REGION Network 3: Перше слово повідомлень
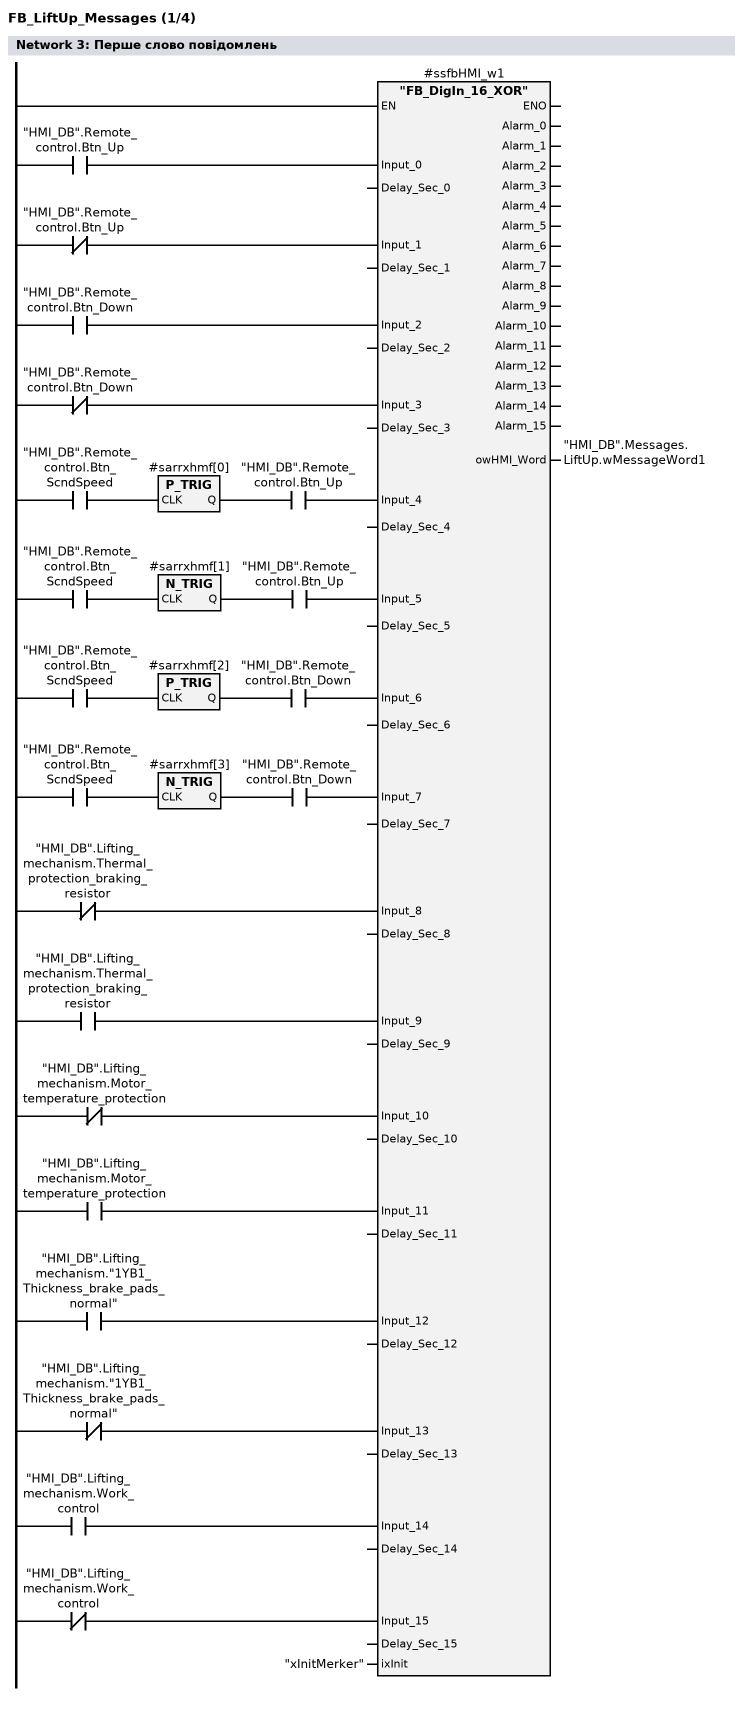
   RUNG wire#powerrail
      #ssfbHMI_w1(Input_0 := wire#w1, Input_1 := wire#w2, Input_2 := wire#w3, Input_3 := wire#w4, Input_4 := wire#w5, Input_5 := wire#w6, Input_6 := wire#w7, Input_7 := wire#w8, Input_8 := wire#w9, Input_9 := wire#w10, Input_10 := wire#w11, Input_11 := wire#w12, Input_12 := wire#w13, Input_13 := wire#w14, Input_14 := wire#w15, Input_15 := wire#w16, Delay_Sec_0 :=, Delay_Sec_1 :=, Delay_Sec_2 :=, Delay_Sec_3 :=, Delay_Sec_4 :=, Delay_Sec_5 :=, Delay_Sec_6 :=, Delay_Sec_7 :=, Delay_Sec_8 :=, Delay_Sec_9 :=, Delay_Sec_10 :=, Delay_Sec_11 :=, Delay_Sec_12 :=, Delay_Sec_13 :=, Delay_Sec_14 :=, Delay_Sec_15 :=, ixInit := "xInitMerker", Alarm_0 =>, Alarm_1 =>, Alarm_2 =>, Alarm_3 =>, Alarm_4 =>, Alarm_5 =>, Alarm_6 =>, Alarm_7 =>, Alarm_8 =>, Alarm_9 =>, Alarm_10 =>, Alarm_11 =>, Alarm_12 =>, Alarm_13 =>, Alarm_14 =>, Alarm_15 =>, owHMI_Word => "HMI_DB".Messages.LiftUp.wMessageWord1)
   END_RUNG
   RUNG wire#powerrail
      Contact( "HMI_DB".Remote_control.Btn_Up )
   END_RUNG wire#w1
   RUNG wire#powerrail
      I_Contact( "HMI_DB".Remote_control.Btn_Up )
   END_RUNG wire#w2
   RUNG wire#powerrail
      Contact( "HMI_DB".Remote_control.Btn_Down )
   END_RUNG wire#w3
   RUNG wire#powerrail
      I_Contact( "HMI_DB".Remote_control.Btn_Down )
   END_RUNG wire#w4
   RUNG wire#powerrail
      Contact( "HMI_DB".Remote_control.Btn_ScndSpeed )
      P_Trig( #sarrxhmf[0] )
      Contact( "HMI_DB".Remote_control.Btn_Up )
   END_RUNG wire#w5
   RUNG wire#powerrail
      Contact( "HMI_DB".Remote_control.Btn_ScndSpeed )
      N_Trig( #sarrxhmf[1] )
      Contact( "HMI_DB".Remote_control.Btn_Up )
   END_RUNG wire#w6
   RUNG wire#powerrail
      Contact( "HMI_DB".Remote_control.Btn_ScndSpeed )
      P_Trig( #sarrxhmf[2] )
      Contact( "HMI_DB".Remote_control.Btn_Down )
   END_RUNG wire#w7
   RUNG wire#powerrail
      Contact( "HMI_DB".Remote_control.Btn_ScndSpeed )
      N_Trig( #sarrxhmf[3] )
      Contact( "HMI_DB".Remote_control.Btn_Down )
   END_RUNG wire#w8
   RUNG wire#powerrail
      I_Contact( "HMI_DB".Lifting_mechanism.Thermal_protection_braking_resistor )
   END_RUNG wire#w9
   RUNG wire#powerrail
      Contact( "HMI_DB".Lifting_mechanism.Thermal_protection_braking_resistor )
   END_RUNG wire#w10
   RUNG wire#powerrail
      I_Contact( "HMI_DB".Lifting_mechanism.Motor_temperature_protection )
   END_RUNG wire#w11
   RUNG wire#powerrail
      Contact( "HMI_DB".Lifting_mechanism.Motor_temperature_protection )
   END_RUNG wire#w12
   RUNG wire#powerrail
      Contact( "HMI_DB".Lifting_mechanism."1YB1_Thickness_brake_pads_normal" )
   END_RUNG wire#w13
   RUNG wire#powerrail
      I_Contact( "HMI_DB".Lifting_mechanism."1YB1_Thickness_brake_pads_normal" )
   END_RUNG wire#w14
   RUNG wire#powerrail
      Contact( "HMI_DB".Lifting_mechanism.Work_control )
   END_RUNG wire#w15
   RUNG wire#powerrail
      I_Contact( "HMI_DB".Lifting_mechanism.Work_control )
   END_RUNG wire#w16
   // the same network as SCL:
   #_w1 := "HMI_DB".Remote_control.Btn_ScndSpeed AND NOT #sarrxhmf[0];   // rising edge
   #sarrxhmf[0] := "HMI_DB".Remote_control.Btn_ScndSpeed;
   #_w2 := NOT "HMI_DB".Remote_control.Btn_ScndSpeed AND #sarrxhmf[1];   // falling edge
   #sarrxhmf[1] := "HMI_DB".Remote_control.Btn_ScndSpeed;
   #_w3 := "HMI_DB".Remote_control.Btn_ScndSpeed AND NOT #sarrxhmf[2];   // rising edge
   #sarrxhmf[2] := "HMI_DB".Remote_control.Btn_ScndSpeed;
   #_w4 := NOT "HMI_DB".Remote_control.Btn_ScndSpeed AND #sarrxhmf[3];   // falling edge
   #sarrxhmf[3] := "HMI_DB".Remote_control.Btn_ScndSpeed;
   #ssfbHMI_w1(Input_0 := "HMI_DB".Remote_control.Btn_Up,   // "FB_DigIn_16_XOR"
               Input_1 := NOT "HMI_DB".Remote_control.Btn_Up,
               Input_2 := "HMI_DB".Remote_control.Btn_Down,
               Input_3 := NOT "HMI_DB".Remote_control.Btn_Down,
               Input_4 := #_w1 AND "HMI_DB".Remote_control.Btn_Up,
               Input_5 := #_w2 AND "HMI_DB".Remote_control.Btn_Up,
               Input_6 := #_w3 AND "HMI_DB".Remote_control.Btn_Down,
               Input_7 := #_w4 AND "HMI_DB".Remote_control.Btn_Down,
               Input_8 := NOT "HMI_DB".Lifting_mechanism.Thermal_protection_braking_resistor,
               Input_9 := "HMI_DB".Lifting_mechanism.Thermal_protection_braking_resistor,
               Input_10 := NOT "HMI_DB".Lifting_mechanism.Motor_temperature_protection,
               Input_11 := "HMI_DB".Lifting_mechanism.Motor_temperature_protection,
               Input_12 := "HMI_DB".Lifting_mechanism."1YB1_Thickness_brake_pads_normal",
               Input_13 := NOT "HMI_DB".Lifting_mechanism."1YB1_Thickness_brake_pads_normal",
               Input_14 := "HMI_DB".Lifting_mechanism.Work_control,
               Input_15 := NOT "HMI_DB".Lifting_mechanism.Work_control,
               ixInit := "xInitMerker",
               owHMI_Word => "HMI_DB".Messages.LiftUp.wMessageWord1);
END_REGION

REGION Network 4: Друге слово повідомлень
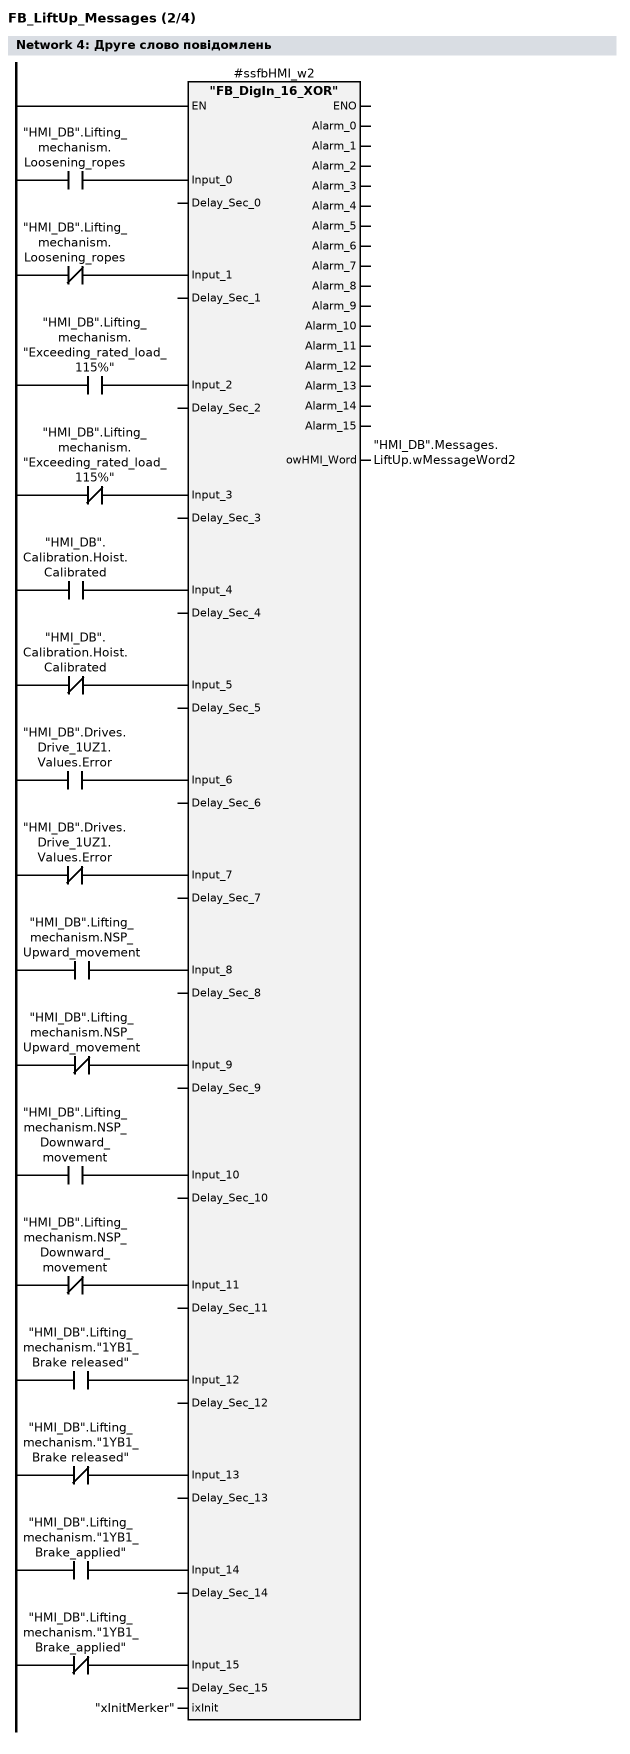
   RUNG wire#powerrail
      #ssfbHMI_w2(Input_0 := wire#w1, Input_1 := wire#w2, Input_2 := wire#w3, Input_3 := wire#w4, Input_4 := wire#w5, Input_5 := wire#w6, Input_6 := wire#w7, Input_7 := wire#w8, Input_8 := wire#w9, Input_9 := wire#w10, Input_10 := wire#w11, Input_11 := wire#w12, Input_12 := wire#w13, Input_13 := wire#w14, Input_14 := wire#w15, Input_15 := wire#w16, Delay_Sec_0 :=, Delay_Sec_1 :=, Delay_Sec_2 :=, Delay_Sec_3 :=, Delay_Sec_4 :=, Delay_Sec_5 :=, Delay_Sec_6 :=, Delay_Sec_7 :=, Delay_Sec_8 :=, Delay_Sec_9 :=, Delay_Sec_10 :=, Delay_Sec_11 :=, Delay_Sec_12 :=, Delay_Sec_13 :=, Delay_Sec_14 :=, Delay_Sec_15 :=, ixInit := "xInitMerker", Alarm_0 =>, Alarm_1 =>, Alarm_2 =>, Alarm_3 =>, Alarm_4 =>, Alarm_5 =>, Alarm_6 =>, Alarm_7 =>, Alarm_8 =>, Alarm_9 =>, Alarm_10 =>, Alarm_11 =>, Alarm_12 =>, Alarm_13 =>, Alarm_14 =>, Alarm_15 =>, owHMI_Word => "HMI_DB".Messages.LiftUp.wMessageWord2)
   END_RUNG
   RUNG wire#powerrail
      Contact( "HMI_DB".Lifting_mechanism.Loosening_ropes )
   END_RUNG wire#w1
   RUNG wire#powerrail
      I_Contact( "HMI_DB".Lifting_mechanism.Loosening_ropes )
   END_RUNG wire#w2
   RUNG wire#powerrail
      Contact( "HMI_DB".Lifting_mechanism."Exceeding_rated_load_115%" )
   END_RUNG wire#w3
   RUNG wire#powerrail
      I_Contact( "HMI_DB".Lifting_mechanism."Exceeding_rated_load_115%" )
   END_RUNG wire#w4
   RUNG wire#powerrail
      Contact( "HMI_DB".Calibration.Hoist.Calibrated )
   END_RUNG wire#w5
   RUNG wire#powerrail
      I_Contact( "HMI_DB".Calibration.Hoist.Calibrated )
   END_RUNG wire#w6
   RUNG wire#powerrail
      Contact( "HMI_DB".Drives.Drive_1UZ1.Values.Error )
   END_RUNG wire#w7
   RUNG wire#powerrail
      I_Contact( "HMI_DB".Drives.Drive_1UZ1.Values.Error )
   END_RUNG wire#w8
   RUNG wire#powerrail
      Contact( "HMI_DB".Lifting_mechanism.NSP_Upward_movement )
   END_RUNG wire#w9
   RUNG wire#powerrail
      I_Contact( "HMI_DB".Lifting_mechanism.NSP_Upward_movement )
   END_RUNG wire#w10
   RUNG wire#powerrail
      Contact( "HMI_DB".Lifting_mechanism.NSP_Downward_movement )
   END_RUNG wire#w11
   RUNG wire#powerrail
      I_Contact( "HMI_DB".Lifting_mechanism.NSP_Downward_movement )
   END_RUNG wire#w12
   RUNG wire#powerrail
      Contact( "HMI_DB".Lifting_mechanism."1YB1_Brake released" )
   END_RUNG wire#w13
   RUNG wire#powerrail
      I_Contact( "HMI_DB".Lifting_mechanism."1YB1_Brake released" )
   END_RUNG wire#w14
   RUNG wire#powerrail
      Contact( "HMI_DB".Lifting_mechanism."1YB1_Brake_applied" )
   END_RUNG wire#w15
   RUNG wire#powerrail
      I_Contact( "HMI_DB".Lifting_mechanism."1YB1_Brake_applied" )
   END_RUNG wire#w16
   // the same network as SCL:
   #ssfbHMI_w2(Input_0 := "HMI_DB".Lifting_mechanism.Loosening_ropes,   // "FB_DigIn_16_XOR"
               Input_1 := NOT "HMI_DB".Lifting_mechanism.Loosening_ropes,
               Input_2 := "HMI_DB".Lifting_mechanism."Exceeding_rated_load_115%",
               Input_3 := NOT "HMI_DB".Lifting_mechanism."Exceeding_rated_load_115%",
               Input_4 := "HMI_DB".Calibration.Hoist.Calibrated,
               Input_5 := NOT "HMI_DB".Calibration.Hoist.Calibrated,
               Input_6 := "HMI_DB".Drives.Drive_1UZ1.Values.Error,
               Input_7 := NOT "HMI_DB".Drives.Drive_1UZ1.Values.Error,
               Input_8 := "HMI_DB".Lifting_mechanism.NSP_Upward_movement,
               Input_9 := NOT "HMI_DB".Lifting_mechanism.NSP_Upward_movement,
               Input_10 := "HMI_DB".Lifting_mechanism.NSP_Downward_movement,
               Input_11 := NOT "HMI_DB".Lifting_mechanism.NSP_Downward_movement,
               Input_12 := "HMI_DB".Lifting_mechanism."1YB1_Brake released",
               Input_13 := NOT "HMI_DB".Lifting_mechanism."1YB1_Brake released",
               Input_14 := "HMI_DB".Lifting_mechanism."1YB1_Brake_applied",
               Input_15 := NOT "HMI_DB".Lifting_mechanism."1YB1_Brake_applied",
               ixInit := "xInitMerker",
               owHMI_Word => "HMI_DB".Messages.LiftUp.wMessageWord2);
END_REGION

REGION Network 5: Третє слово повідомлень
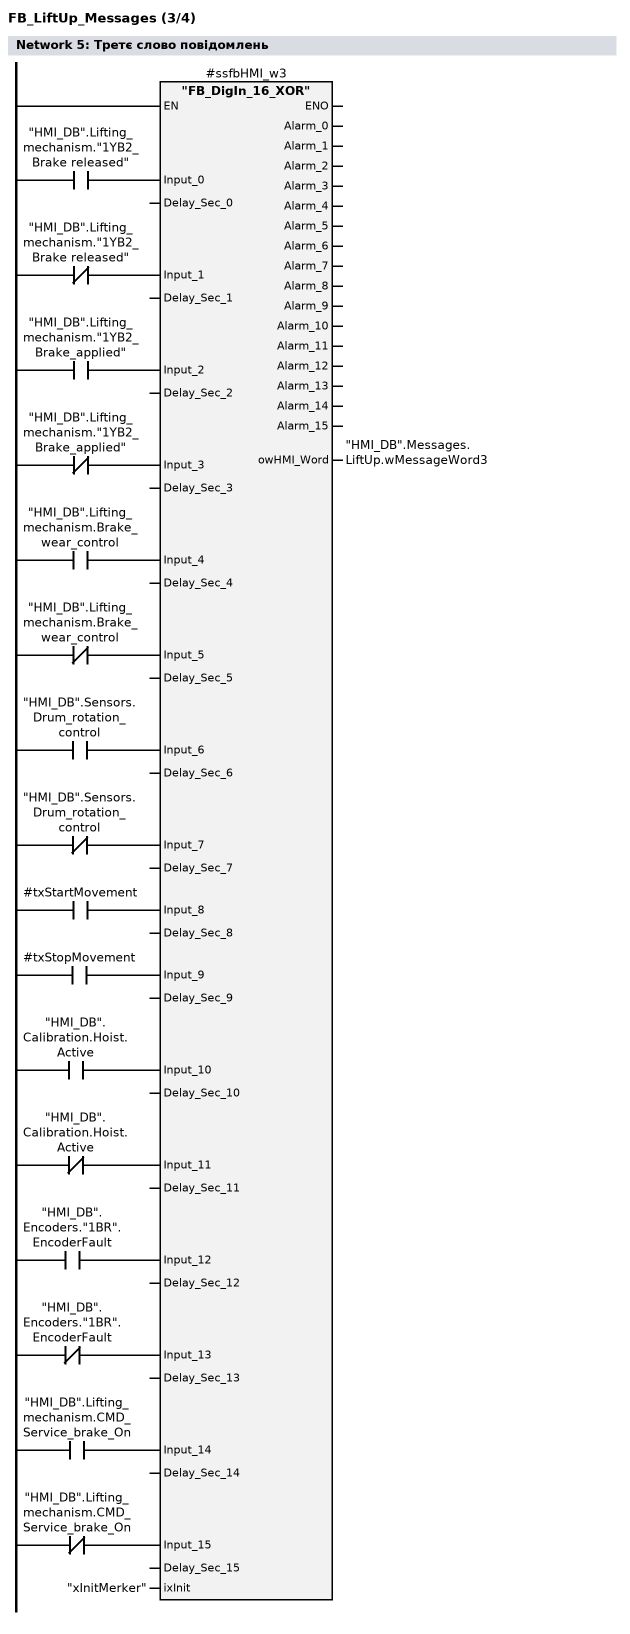
   RUNG wire#powerrail
      #ssfbHMI_w3(Input_0 := wire#w1, Input_1 := wire#w2, Input_2 := wire#w3, Input_3 := wire#w4, Input_4 := wire#w5, Input_5 := wire#w6, Input_6 := wire#w7, Input_7 := wire#w8, Input_8 := wire#w9, Input_9 := wire#w10, Input_10 := wire#w11, Input_11 := wire#w12, Input_12 := wire#w13, Input_13 := wire#w14, Input_14 := wire#w15, Input_15 := wire#w16, Delay_Sec_0 :=, Delay_Sec_1 :=, Delay_Sec_2 :=, Delay_Sec_3 :=, Delay_Sec_4 :=, Delay_Sec_5 :=, Delay_Sec_6 :=, Delay_Sec_7 :=, Delay_Sec_8 :=, Delay_Sec_9 :=, Delay_Sec_10 :=, Delay_Sec_11 :=, Delay_Sec_12 :=, Delay_Sec_13 :=, Delay_Sec_14 :=, Delay_Sec_15 :=, ixInit := "xInitMerker", Alarm_0 =>, Alarm_1 =>, Alarm_2 =>, Alarm_3 =>, Alarm_4 =>, Alarm_5 =>, Alarm_6 =>, Alarm_7 =>, Alarm_8 =>, Alarm_9 =>, Alarm_10 =>, Alarm_11 =>, Alarm_12 =>, Alarm_13 =>, Alarm_14 =>, Alarm_15 =>, owHMI_Word => "HMI_DB".Messages.LiftUp.wMessageWord3)
   END_RUNG
   RUNG wire#powerrail
      Contact( "HMI_DB".Lifting_mechanism."1YB2_Brake released" )
   END_RUNG wire#w1
   RUNG wire#powerrail
      I_Contact( "HMI_DB".Lifting_mechanism."1YB2_Brake released" )
   END_RUNG wire#w2
   RUNG wire#powerrail
      Contact( "HMI_DB".Lifting_mechanism."1YB2_Brake_applied" )
   END_RUNG wire#w3
   RUNG wire#powerrail
      I_Contact( "HMI_DB".Lifting_mechanism."1YB2_Brake_applied" )
   END_RUNG wire#w4
   RUNG wire#powerrail
      Contact( "HMI_DB".Lifting_mechanism.Brake_wear_control )
   END_RUNG wire#w5
   RUNG wire#powerrail
      I_Contact( "HMI_DB".Lifting_mechanism.Brake_wear_control )
   END_RUNG wire#w6
   RUNG wire#powerrail
      Contact( "HMI_DB".Sensors.Drum_rotation_control )
   END_RUNG wire#w7
   RUNG wire#powerrail
      I_Contact( "HMI_DB".Sensors.Drum_rotation_control )
   END_RUNG wire#w8
   RUNG wire#powerrail
      Contact( #txStartMovement )
   END_RUNG wire#w9
   RUNG wire#powerrail
      Contact( #txStopMovement )
   END_RUNG wire#w10
   RUNG wire#powerrail
      Contact( "HMI_DB".Calibration.Hoist.Active )
   END_RUNG wire#w11
   RUNG wire#powerrail
      I_Contact( "HMI_DB".Calibration.Hoist.Active )
   END_RUNG wire#w12
   RUNG wire#powerrail
      Contact( "HMI_DB".Encoders."1BR".EncoderFault )
   END_RUNG wire#w13
   RUNG wire#powerrail
      I_Contact( "HMI_DB".Encoders."1BR".EncoderFault )
   END_RUNG wire#w14
   RUNG wire#powerrail
      Contact( "HMI_DB".Lifting_mechanism.CMD_Service_brake_On )
   END_RUNG wire#w15
   RUNG wire#powerrail
      I_Contact( "HMI_DB".Lifting_mechanism.CMD_Service_brake_On )
   END_RUNG wire#w16
   // the same network as SCL:
   #ssfbHMI_w3(Input_0 := "HMI_DB".Lifting_mechanism."1YB2_Brake released",   // "FB_DigIn_16_XOR"
               Input_1 := NOT "HMI_DB".Lifting_mechanism."1YB2_Brake released",
               Input_2 := "HMI_DB".Lifting_mechanism."1YB2_Brake_applied",
               Input_3 := NOT "HMI_DB".Lifting_mechanism."1YB2_Brake_applied",
               Input_4 := "HMI_DB".Lifting_mechanism.Brake_wear_control,
               Input_5 := NOT "HMI_DB".Lifting_mechanism.Brake_wear_control,
               Input_6 := "HMI_DB".Sensors.Drum_rotation_control,
               Input_7 := NOT "HMI_DB".Sensors.Drum_rotation_control,
               Input_8 := #txStartMovement,
               Input_9 := #txStopMovement,
               Input_10 := "HMI_DB".Calibration.Hoist.Active,
               Input_11 := NOT "HMI_DB".Calibration.Hoist.Active,
               Input_12 := "HMI_DB".Encoders."1BR".EncoderFault,
               Input_13 := NOT "HMI_DB".Encoders."1BR".EncoderFault,
               Input_14 := "HMI_DB".Lifting_mechanism.CMD_Service_brake_On,
               Input_15 := NOT "HMI_DB".Lifting_mechanism.CMD_Service_brake_On,
               ixInit := "xInitMerker",
               owHMI_Word => "HMI_DB".Messages.LiftUp.wMessageWord3);
END_REGION

REGION Network 6: Четверте слово повідомлень
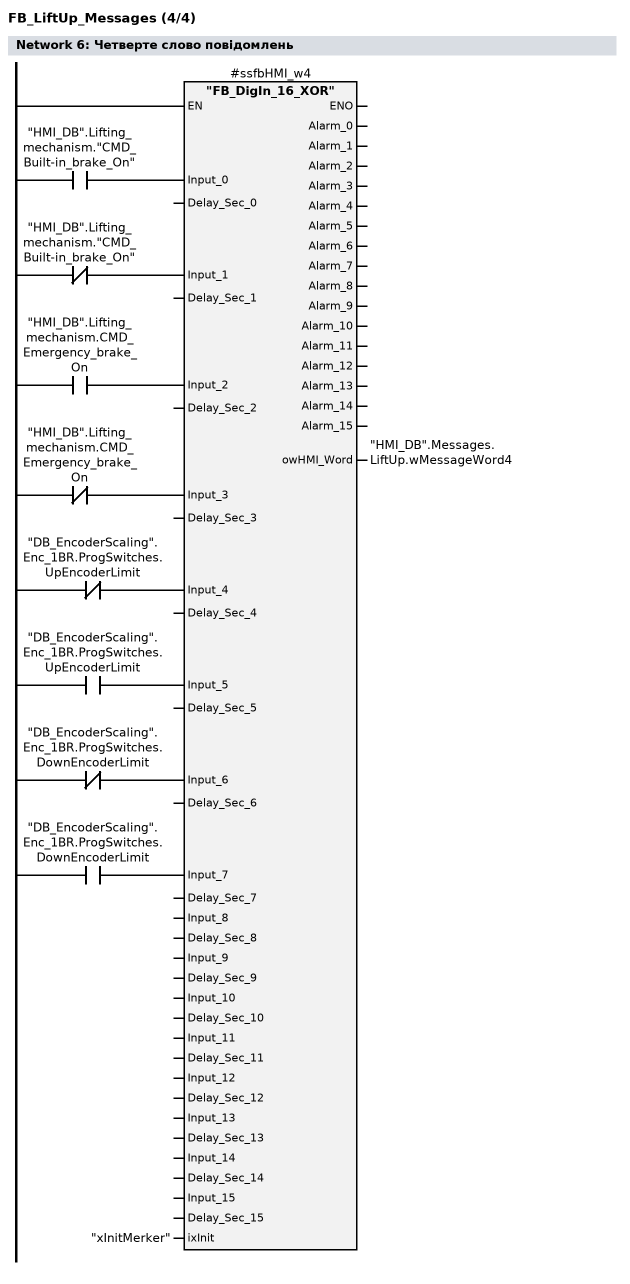
   RUNG wire#powerrail
      #ssfbHMI_w4(Input_0 := wire#w1, Input_1 := wire#w2, Input_2 := wire#w3, Input_3 := wire#w4, Input_4 := wire#w5, Input_5 := wire#w6, Input_6 := wire#w7, Input_7 := wire#w8, Delay_Sec_0 :=, Delay_Sec_1 :=, Delay_Sec_2 :=, Delay_Sec_3 :=, Delay_Sec_4 :=, Delay_Sec_5 :=, Delay_Sec_6 :=, Delay_Sec_7 :=, Input_8 :=, Delay_Sec_8 :=, Input_9 :=, Delay_Sec_9 :=, Input_10 :=, Delay_Sec_10 :=, Input_11 :=, Delay_Sec_11 :=, Input_12 :=, Delay_Sec_12 :=, Input_13 :=, Delay_Sec_13 :=, Input_14 :=, Delay_Sec_14 :=, Input_15 :=, Delay_Sec_15 :=, ixInit := "xInitMerker", Alarm_0 =>, Alarm_1 =>, Alarm_2 =>, Alarm_3 =>, Alarm_4 =>, Alarm_5 =>, Alarm_6 =>, Alarm_7 =>, Alarm_8 =>, Alarm_9 =>, Alarm_10 =>, Alarm_11 =>, Alarm_12 =>, Alarm_13 =>, Alarm_14 =>, Alarm_15 =>, owHMI_Word => "HMI_DB".Messages.LiftUp.wMessageWord4)
   END_RUNG
   RUNG wire#powerrail
      Contact( "HMI_DB".Lifting_mechanism."CMD_Built-in_brake_On" )
   END_RUNG wire#w1
   RUNG wire#powerrail
      I_Contact( "HMI_DB".Lifting_mechanism."CMD_Built-in_brake_On" )
   END_RUNG wire#w2
   RUNG wire#powerrail
      Contact( "HMI_DB".Lifting_mechanism.CMD_Emergency_brake_On )
   END_RUNG wire#w3
   RUNG wire#powerrail
      I_Contact( "HMI_DB".Lifting_mechanism.CMD_Emergency_brake_On )
   END_RUNG wire#w4
   RUNG wire#powerrail
      I_Contact( "DB_EncoderScaling".Enc_1BR.ProgSwitches.UpEncoderLimit )
   END_RUNG wire#w5
   RUNG wire#powerrail
      Contact( "DB_EncoderScaling".Enc_1BR.ProgSwitches.UpEncoderLimit )
   END_RUNG wire#w6
   RUNG wire#powerrail
      I_Contact( "DB_EncoderScaling".Enc_1BR.ProgSwitches.DownEncoderLimit )
   END_RUNG wire#w7
   RUNG wire#powerrail
      Contact( "DB_EncoderScaling".Enc_1BR.ProgSwitches.DownEncoderLimit )
   END_RUNG wire#w8
   // the same network as SCL:
   #ssfbHMI_w4(Input_0 := "HMI_DB".Lifting_mechanism."CMD_Built-in_brake_On",   // "FB_DigIn_16_XOR"
               Input_1 := NOT "HMI_DB".Lifting_mechanism."CMD_Built-in_brake_On",
               Input_2 := "HMI_DB".Lifting_mechanism.CMD_Emergency_brake_On,
               Input_3 := NOT "HMI_DB".Lifting_mechanism.CMD_Emergency_brake_On,
               Input_4 := NOT "DB_EncoderScaling".Enc_1BR.ProgSwitches.UpEncoderLimit,
               Input_5 := "DB_EncoderScaling".Enc_1BR.ProgSwitches.UpEncoderLimit,
               Input_6 := NOT "DB_EncoderScaling".Enc_1BR.ProgSwitches.DownEncoderLimit,
               Input_7 := "DB_EncoderScaling".Enc_1BR.ProgSwitches.DownEncoderLimit,
               ixInit := "xInitMerker",
               owHMI_Word => "HMI_DB".Messages.LiftUp.wMessageWord4);
END_REGION
END_FUNCTION_BLOCK

FUNCTION "FC_Lifting" : Void   // FC300, LAD
{ S7_Optimized_Access := 'TRUE' }
VERSION : 0.1
   VAR_TEMP   // added for the SCL form of the ladder/FBD networks
      _w1 : Bool;
   END_VAR
BEGIN

REGION Network 2: =================Блокування пристрою ручного керування========================
END_REGION

REGION Network 3: Механізм підйому. Вимикачі кінцеві на гальмі 1YB2. Дозвіл роботи (MPP роз'єднаний з гальмом)
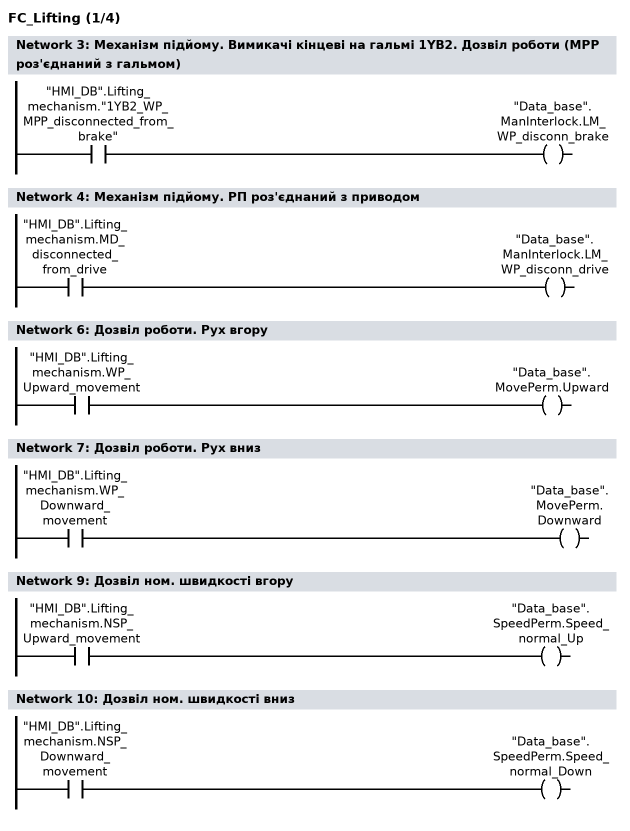
   RUNG wire#powerrail
      Contact( "HMI_DB".Lifting_mechanism."1YB2_WP_MPP_disconnected_from_brake" )
      Coil( "Data_base".ManInterlock.LM_WP_disconn_brake )
   END_RUNG
   // the same network as SCL:
   "Data_base".ManInterlock.LM_WP_disconn_brake := "HMI_DB".Lifting_mechanism."1YB2_WP_MPP_disconnected_from_brake";
END_REGION

REGION Network 4: Механізм підйому. РП роз'єднаний з приводом
   RUNG wire#powerrail
      Contact( "HMI_DB".Lifting_mechanism.MD_disconnected_from_drive )
      Coil( "Data_base".ManInterlock.LM_WP_disconn_drive )
   END_RUNG
   // the same network as SCL:
   "Data_base".ManInterlock.LM_WP_disconn_drive := "HMI_DB".Lifting_mechanism.MD_disconnected_from_drive;
END_REGION

REGION Network 5: ================Дозвіл роботи====================
END_REGION

REGION Network 6: Дозвіл роботи. Рух вгору
   RUNG wire#powerrail
      Contact( "HMI_DB".Lifting_mechanism.WP_Upward_movement )
      Coil( "Data_base".MovePerm.Upward )
   END_RUNG
   // the same network as SCL:
   "Data_base".MovePerm.Upward := "HMI_DB".Lifting_mechanism.WP_Upward_movement;
END_REGION

REGION Network 7: Дозвіл роботи. Рух вниз
   RUNG wire#powerrail
      Contact( "HMI_DB".Lifting_mechanism.WP_Downward_movement )
      Coil( "Data_base".MovePerm.Downward )
   END_RUNG
   // the same network as SCL:
   "Data_base".MovePerm.Downward := "HMI_DB".Lifting_mechanism.WP_Downward_movement;
END_REGION

REGION Network 8: ================Дозвіл нормальної швидкості =================
END_REGION

REGION Network 9: Дозвіл ном. швидкості вгору
   RUNG wire#powerrail
      Contact( "HMI_DB".Lifting_mechanism.NSP_Upward_movement )
      Coil( "Data_base".SpeedPerm.Speed_normal_Up )
   END_RUNG
   // the same network as SCL:
   "Data_base".SpeedPerm.Speed_normal_Up := "HMI_DB".Lifting_mechanism.NSP_Upward_movement;
END_REGION

REGION Network 10: Дозвіл ном. швидкості вниз
   RUNG wire#powerrail
      Contact( "HMI_DB".Lifting_mechanism.NSP_Downward_movement )
      Coil( "Data_base".SpeedPerm.Speed_normal_Down )
   END_RUNG
   // the same network as SCL:
   "Data_base".SpeedPerm.Speed_normal_Down := "HMI_DB".Lifting_mechanism.NSP_Downward_movement;
END_REGION

REGION Network 11: ===============Керування механізмом підйому================
END_REGION

REGION Network 12: Механізм підйому
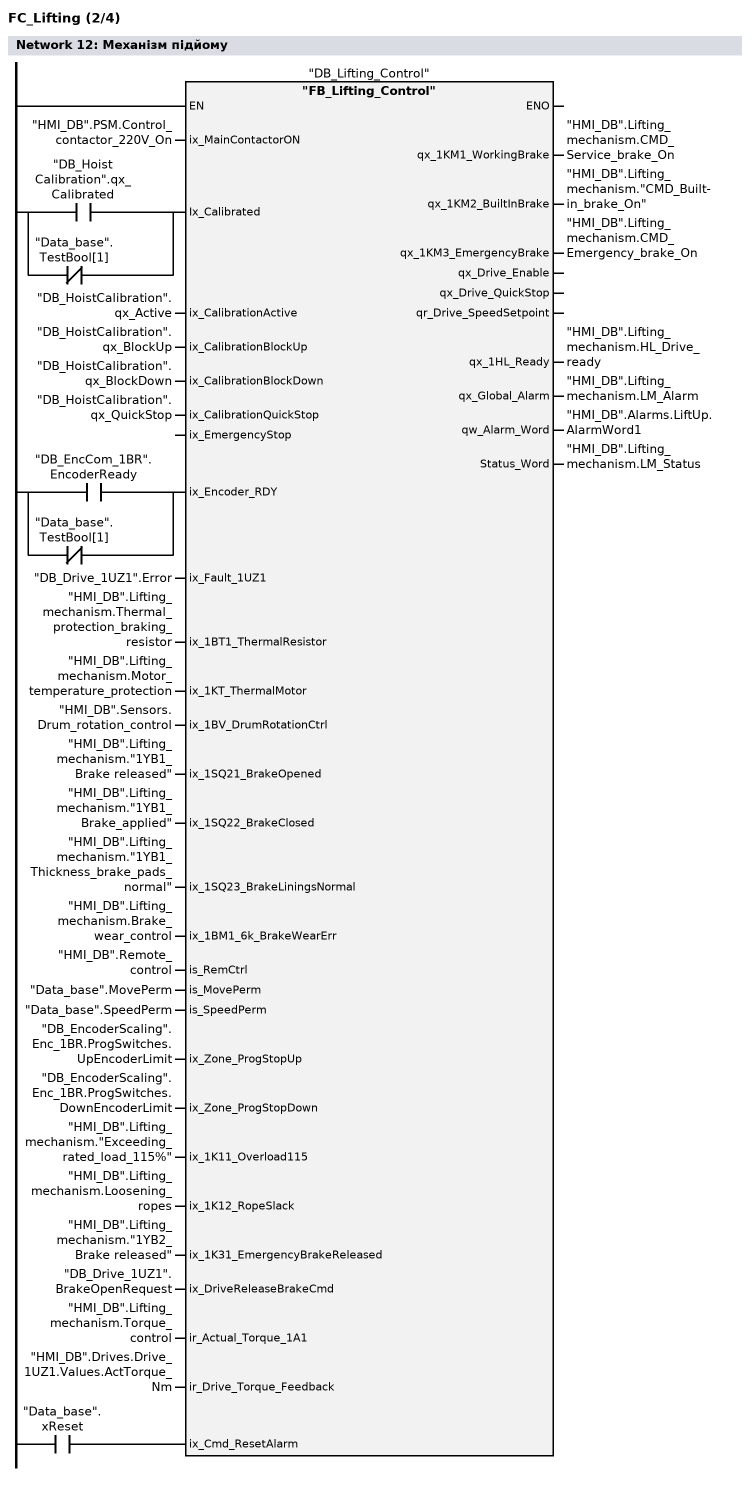
   RUNG wire#powerrail
      "DB_Lifting_Control"(Ix_Calibrated := wire#w1, ix_Encoder_RDY := wire#w2, ix_Cmd_ResetAlarm := wire#w3, ix_MainContactorON := "HMI_DB".PSM.Control_contactor_220V_On, ix_CalibrationActive := "DB_HoistCalibration".qx_Active, ix_CalibrationBlockUp := "DB_HoistCalibration".qx_BlockUp, ix_CalibrationBlockDown := "DB_HoistCalibration".qx_BlockDown, ix_CalibrationQuickStop := "DB_HoistCalibration".qx_QuickStop, ix_EmergencyStop :=, ix_Fault_1UZ1 := "DB_Drive_1UZ1".Error, ix_1BT1_ThermalResistor := "HMI_DB".Lifting_mechanism.Thermal_protection_braking_resistor, ix_1KT_ThermalMotor := "HMI_DB".Lifting_mechanism.Motor_temperature_protection, ix_1BV_DrumRotationCtrl := "HMI_DB".Sensors.Drum_rotation_control, ix_1SQ21_BrakeOpened := "HMI_DB".Lifting_mechanism."1YB1_Brake released", ix_1SQ22_BrakeClosed := "HMI_DB".Lifting_mechanism."1YB1_Brake_applied", ix_1SQ23_BrakeLiningsNormal := "HMI_DB".Lifting_mechanism."1YB1_Thickness_brake_pads_normal", ix_1BM1_6k_BrakeWearErr := "HMI_DB".Lifting_mechanism.Brake_wear_control, is_RemCtrl := "HMI_DB".Remote_control, is_MovePerm := "Data_base".MovePerm, is_SpeedPerm := "Data_base".SpeedPerm, ix_Zone_ProgStopUp := "DB_EncoderScaling".Enc_1BR.ProgSwitches.UpEncoderLimit, ix_Zone_ProgStopDown := "DB_EncoderScaling".Enc_1BR.ProgSwitches.DownEncoderLimit, ix_1K11_Overload115 := "HMI_DB".Lifting_mechanism."Exceeding_rated_load_115%", ix_1K12_RopeSlack := "HMI_DB".Lifting_mechanism.Loosening_ropes, ix_1K31_EmergencyBrakeReleased := "HMI_DB".Lifting_mechanism."1YB2_Brake released", ix_DriveReleaseBrakeCmd := "DB_Drive_1UZ1".BrakeOpenRequest, ir_Actual_Torque_1A1 := "HMI_DB".Lifting_mechanism.Torque_control, ir_Drive_Torque_Feedback := "HMI_DB".Drives.Drive_1UZ1.Values.ActTorque_Nm, qx_1KM1_WorkingBrake => "HMI_DB".Lifting_mechanism.CMD_Service_brake_On, qx_1KM2_BuiltInBrake => "HMI_DB".Lifting_mechanism."CMD_Built-in_brake_On", qx_1KM3_EmergencyBrake => "HMI_DB".Lifting_mechanism.CMD_Emergency_brake_On, qx_Drive_Enable =>, qx_Drive_QuickStop =>, qr_Drive_SpeedSetpoint =>, qx_1HL_Ready => "HMI_DB".Lifting_mechanism.HL_Drive_ready, qx_Global_Alarm => "HMI_DB".Lifting_mechanism.LM_Alarm, qw_Alarm_Word => "HMI_DB".Alarms.LiftUp.AlarmWord1, Status_Word => "HMI_DB".Lifting_mechanism.LM_Status)
   END_RUNG
   RUNG wire#powerrail
      Contact( "DB_HoistCalibration".qx_Calibrated )
   END_RUNG wire#w1
   RUNG wire#powerrail
      I_Contact( "Data_base".TestBool[1] )
   END_RUNG wire#w1
   RUNG wire#powerrail
      Contact( "DB_EncCom_1BR".EncoderReady )
   END_RUNG wire#w2
   RUNG wire#powerrail
      I_Contact( "Data_base".TestBool[1] )
   END_RUNG wire#w2
   RUNG wire#powerrail
      Contact( "Data_base".xReset )
   END_RUNG wire#w3
   // the same network as SCL:
   "DB_Lifting_Control"(ix_MainContactorON := "HMI_DB".PSM.Control_contactor_220V_On,   // "FB_Lifting_Control"
                        Ix_Calibrated := "DB_HoistCalibration".qx_Calibrated OR NOT "Data_base".TestBool[1],
                        ix_CalibrationActive := "DB_HoistCalibration".qx_Active,
                        ix_CalibrationBlockUp := "DB_HoistCalibration".qx_BlockUp,
                        ix_CalibrationBlockDown := "DB_HoistCalibration".qx_BlockDown,
                        ix_CalibrationQuickStop := "DB_HoistCalibration".qx_QuickStop,
                        ix_Encoder_RDY := "DB_EncCom_1BR".EncoderReady OR NOT "Data_base".TestBool[1],
                        ix_Fault_1UZ1 := "DB_Drive_1UZ1".Error,
                        ix_1BT1_ThermalResistor := "HMI_DB".Lifting_mechanism.Thermal_protection_braking_resistor,
                        ix_1KT_ThermalMotor := "HMI_DB".Lifting_mechanism.Motor_temperature_protection,
                        ix_1BV_DrumRotationCtrl := "HMI_DB".Sensors.Drum_rotation_control,
                        ix_1SQ21_BrakeOpened := "HMI_DB".Lifting_mechanism."1YB1_Brake released",
                        ix_1SQ22_BrakeClosed := "HMI_DB".Lifting_mechanism."1YB1_Brake_applied",
                        ix_1SQ23_BrakeLiningsNormal := "HMI_DB".Lifting_mechanism."1YB1_Thickness_brake_pads_normal",
                        ix_1BM1_6k_BrakeWearErr := "HMI_DB".Lifting_mechanism.Brake_wear_control,
                        is_RemCtrl := "HMI_DB".Remote_control,
                        is_MovePerm := "Data_base".MovePerm,
                        is_SpeedPerm := "Data_base".SpeedPerm,
                        ix_Zone_ProgStopUp := "DB_EncoderScaling".Enc_1BR.ProgSwitches.UpEncoderLimit,
                        ix_Zone_ProgStopDown := "DB_EncoderScaling".Enc_1BR.ProgSwitches.DownEncoderLimit,
                        ix_1K11_Overload115 := "HMI_DB".Lifting_mechanism."Exceeding_rated_load_115%",
                        ix_1K12_RopeSlack := "HMI_DB".Lifting_mechanism.Loosening_ropes,
                        ix_1K31_EmergencyBrakeReleased := "HMI_DB".Lifting_mechanism."1YB2_Brake released",
                        ix_DriveReleaseBrakeCmd := "DB_Drive_1UZ1".BrakeOpenRequest,
                        ir_Actual_Torque_1A1 := "HMI_DB".Lifting_mechanism.Torque_control,
                        ir_Drive_Torque_Feedback := "HMI_DB".Drives.Drive_1UZ1.Values.ActTorque_Nm,
                        ix_Cmd_ResetAlarm := "Data_base".xReset,
                        qx_1KM1_WorkingBrake => "HMI_DB".Lifting_mechanism.CMD_Service_brake_On,
                        qx_1KM2_BuiltInBrake => "HMI_DB".Lifting_mechanism."CMD_Built-in_brake_On",
                        qx_1KM3_EmergencyBrake => "HMI_DB".Lifting_mechanism.CMD_Emergency_brake_On,
                        qx_1HL_Ready => "HMI_DB".Lifting_mechanism.HL_Drive_ready,
                        qx_Global_Alarm => "HMI_DB".Lifting_mechanism.LM_Alarm,
                        qw_Alarm_Word => "HMI_DB".Alarms.LiftUp.AlarmWord1,
                        Status_Word => "HMI_DB".Lifting_mechanism.LM_Status);
END_REGION

REGION Network 13: Повідомлення дій оператора
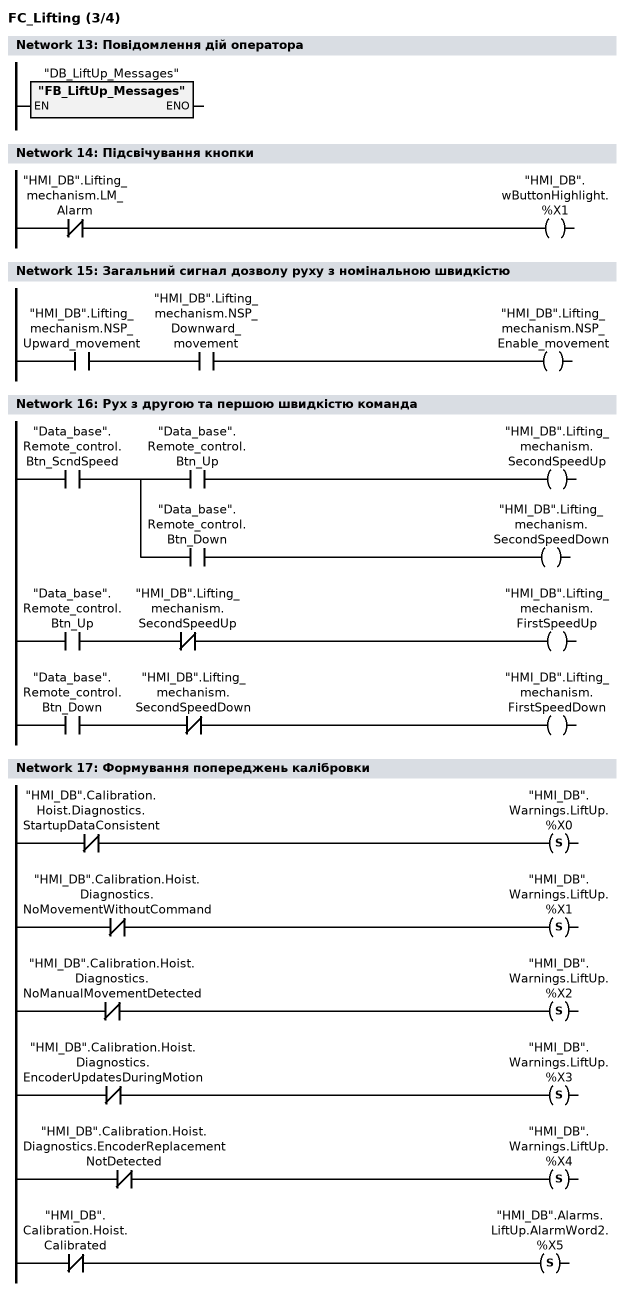
   RUNG wire#powerrail
      "DB_LiftUp_Messages"()
   END_RUNG
   // the same network as SCL:
   "DB_LiftUp_Messages"();   // "FB_LiftUp_Messages"
END_REGION

REGION Network 14: Підсвічування кнопки
   RUNG wire#powerrail
      I_Contact( "HMI_DB".Lifting_mechanism.LM_Alarm )
      Coil( "HMI_DB".wButtonHighlight.%X1 )
   END_RUNG
   // the same network as SCL:
   "HMI_DB".wButtonHighlight.%X1 := NOT "HMI_DB".Lifting_mechanism.LM_Alarm;
END_REGION

REGION Network 15: Загальний сигнал дозволу руху з номінальною швидкістю
   RUNG wire#powerrail
      Contact( "HMI_DB".Lifting_mechanism.NSP_Upward_movement )
      Contact( "HMI_DB".Lifting_mechanism.NSP_Downward_movement )
      Coil( "HMI_DB".Lifting_mechanism.NSP_Enable_movement )
   END_RUNG
   // the same network as SCL:
   "HMI_DB".Lifting_mechanism.NSP_Enable_movement := "HMI_DB".Lifting_mechanism.NSP_Upward_movement AND "HMI_DB".Lifting_mechanism.NSP_Downward_movement;
END_REGION

REGION Network 16: Рух з другою та першою швидкістю команда
   RUNG wire#powerrail
      Contact( "Data_base".Remote_control.Btn_ScndSpeed )
      wire#w1
      Contact( "Data_base".Remote_control.Btn_Up )
      Coil( "HMI_DB".Lifting_mechanism.SecondSpeedUp )
   END_RUNG
   RUNG wire#w1
      Contact( "Data_base".Remote_control.Btn_Down )
      Coil( "HMI_DB".Lifting_mechanism.SecondSpeedDown )
   END_RUNG
   RUNG wire#powerrail
      Contact( "Data_base".Remote_control.Btn_Up )
      I_Contact( "HMI_DB".Lifting_mechanism.SecondSpeedUp )
      Coil( "HMI_DB".Lifting_mechanism.FirstSpeedUp )
   END_RUNG
   RUNG wire#powerrail
      Contact( "Data_base".Remote_control.Btn_Down )
      I_Contact( "HMI_DB".Lifting_mechanism.SecondSpeedDown )
      Coil( "HMI_DB".Lifting_mechanism.FirstSpeedDown )
   END_RUNG
   // the same network as SCL:
   "HMI_DB".Lifting_mechanism.SecondSpeedUp := "Data_base".Remote_control.Btn_ScndSpeed AND "Data_base".Remote_control.Btn_Up;
   "HMI_DB".Lifting_mechanism.SecondSpeedDown := "Data_base".Remote_control.Btn_ScndSpeed AND "Data_base".Remote_control.Btn_Down;
   "HMI_DB".Lifting_mechanism.FirstSpeedUp := "Data_base".Remote_control.Btn_Up AND NOT "HMI_DB".Lifting_mechanism.SecondSpeedUp;
   "HMI_DB".Lifting_mechanism.FirstSpeedDown := "Data_base".Remote_control.Btn_Down AND NOT "HMI_DB".Lifting_mechanism.SecondSpeedDown;
END_REGION

REGION Network 17: Формування попереджень калібровки
   RUNG wire#powerrail
      I_Contact( "HMI_DB".Calibration.Hoist.Diagnostics.StartupDataConsistent )
      S_Coil( "HMI_DB".Warnings.LiftUp.%X0 )
   END_RUNG
   RUNG wire#powerrail
      I_Contact( "HMI_DB".Calibration.Hoist.Diagnostics.NoMovementWithoutCommand )
      S_Coil( "HMI_DB".Warnings.LiftUp.%X1 )
   END_RUNG
   RUNG wire#powerrail
      I_Contact( "HMI_DB".Calibration.Hoist.Diagnostics.NoManualMovementDetected )
      S_Coil( "HMI_DB".Warnings.LiftUp.%X2 )
   END_RUNG
   RUNG wire#powerrail
      I_Contact( "HMI_DB".Calibration.Hoist.Diagnostics.EncoderUpdatesDuringMotion )
      S_Coil( "HMI_DB".Warnings.LiftUp.%X3 )
   END_RUNG
   RUNG wire#powerrail
      I_Contact( "HMI_DB".Calibration.Hoist.Diagnostics.EncoderReplacementNotDetected )
      S_Coil( "HMI_DB".Warnings.LiftUp.%X4 )
   END_RUNG
   RUNG wire#powerrail
      I_Contact( "HMI_DB".Calibration.Hoist.Calibrated )
      S_Coil( "HMI_DB".Alarms.LiftUp.AlarmWord2.%X5 )
   END_RUNG
   // the same network as SCL:
   IF NOT "HMI_DB".Calibration.Hoist.Diagnostics.StartupDataConsistent THEN
       "HMI_DB".Warnings.LiftUp.%X0 := TRUE;
   END_IF;
   IF NOT "HMI_DB".Calibration.Hoist.Diagnostics.NoMovementWithoutCommand THEN
       "HMI_DB".Warnings.LiftUp.%X1 := TRUE;
   END_IF;
   IF NOT "HMI_DB".Calibration.Hoist.Diagnostics.NoManualMovementDetected THEN
       "HMI_DB".Warnings.LiftUp.%X2 := TRUE;
   END_IF;
   IF NOT "HMI_DB".Calibration.Hoist.Diagnostics.EncoderUpdatesDuringMotion THEN
       "HMI_DB".Warnings.LiftUp.%X3 := TRUE;
   END_IF;
   IF NOT "HMI_DB".Calibration.Hoist.Diagnostics.EncoderReplacementNotDetected THEN
       "HMI_DB".Warnings.LiftUp.%X4 := TRUE;
   END_IF;
   IF NOT "HMI_DB".Calibration.Hoist.Calibrated THEN "HMI_DB".Alarms.LiftUp.AlarmWord2.%X5 := TRUE; END_IF;
END_REGION

REGION Network 18: Скидання попереджень калібровки
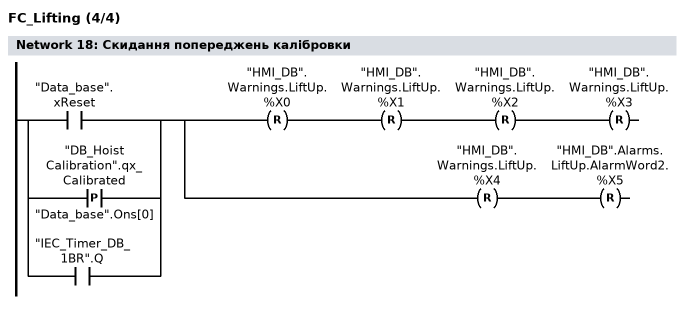
   RUNG wire#powerrail
      Contact( "Data_base".xReset )
      wire#w1
      R_Coil( "HMI_DB".Warnings.LiftUp.%X0 )
      R_Coil( "HMI_DB".Warnings.LiftUp.%X1 )
      R_Coil( "HMI_DB".Warnings.LiftUp.%X2 )
      R_Coil( "HMI_DB".Warnings.LiftUp.%X3 )
   END_RUNG
   RUNG wire#powerrail
      P_Contact(operand := "DB_HoistCalibration".qx_Calibrated, bit := "Data_base".Ons[0])
   END_RUNG wire#w1
   RUNG wire#powerrail
      Contact( "IEC_Timer_DB_1BR".Q )
   END_RUNG wire#w1
   RUNG wire#w1
      R_Coil( "HMI_DB".Warnings.LiftUp.%X4 )
      R_Coil( "HMI_DB".Alarms.LiftUp.AlarmWord2.%X5 )
   END_RUNG
   // the same network as SCL:
   #_w1 := "DB_HoistCalibration".qx_Calibrated AND NOT "Data_base".Ons[0];   // rising edge of "DB_HoistCalibration".qx_Calibrated
   "Data_base".Ons[0] := "DB_HoistCalibration".qx_Calibrated;
   IF "Data_base".xReset OR #_w1 OR "IEC_Timer_DB_1BR".Q THEN
       "HMI_DB".Warnings.LiftUp.%X0 := FALSE;
       "HMI_DB".Warnings.LiftUp.%X1 := FALSE;
       "HMI_DB".Warnings.LiftUp.%X2 := FALSE;
       "HMI_DB".Warnings.LiftUp.%X3 := FALSE;
       "HMI_DB".Warnings.LiftUp.%X4 := FALSE;
       "HMI_DB".Alarms.LiftUp.AlarmWord2.%X5 := FALSE;
   END_IF;
END_REGION
END_FUNCTION

// folder: 400_3UZ1_Trolley_movement(TM)

FUNCTION_BLOCK "FB_Trolley_Control"   // FB400, SCL
{ S7_Optimized_Access := 'TRUE' }
VERSION : 0.1
   VAR_INPUT
      ix_MainContactorON : Bool;   // Головний контактор увімкнено
      ix_Calibrated : Bool;   // Механізм візка калібровано по енкодеру
      ix_CalibrationActive : Bool;   // Активна процедура калібровки візка
      ix_CalibrationBlockForward : Bool;   // Заборона руху вперед від блока калібровки
      ix_CalibrationBlockBackward : Bool;   // Заборона руху назад від блока калібровки
      ix_CalibrationQuickStop : Bool;   // Запит Quick Stop від блока калібровки
      ix_EmergencyStop : Bool;   // Загальний аварійний стоп
      ix_Encoder_RDY : Bool;
      ix_Fault_3UZ1 : Bool;
      ix_2BT1_ThermalResistor : Bool;   // Термостат гальмівного резистора
      ix_2KT_ThermalMotor : Bool;   // Термісторне реле захисту двигуна візка 2M1
      is_RemCtrl : "udtRemCtrl";   // Кнопки руху з пульта (для контролю нульового положення при старті)
      is_MovePerm : "udtMovePerm";   // Кінцеві вимикачі руху крайніх положень
      is_SpeedPerm : "udtSpeedPerm";   // Кінцеві вимикачі швидкості руху
      ix_Zone_ProgStopFwd : Bool;   // Програмна зона зупинки Вперед (по енкодеру)
      ix_Zone_ProgStopBwd : Bool;   // Програмна зона зупинки Назад (по енкодеру)
      ix_Zone_BackPreStop : Bool;   // Візок знаходиться в зоні технологічного передзупину назад
      ix_1K11_Overload115 : Bool;   // Відсутність сигналу = Перевантаження 115%
      ix_DriveReleaseBrakeCmd : Bool;   // Команда розгальмування від ЧП 2UZ1 в телеграмі
      ix_Cmd_ResetAlarm : Bool;   // Кнопка скидання аварій (квітування)
   END_VAR
   VAR_OUTPUT
      qx_2KM1_WorkingBrake : Bool;   // Пускач зовнішнього робочого гальма 2MB1
      qx_Drive_Enable : Bool;   // Один загальний сигнал дозволу руху / роботи ЧП
      qx_Drive_QuickStop : Bool;   // Команда швидкого гальмування Quick Stop
      qr_Drive_SpeedSetpoint : Real;   // Завдання швидкості на ЧП зі знаком
      qx_2HL_Ready : Bool;   // Світловий індикатор готовності візка
      qx_Global_Alarm : Bool;   // Сигнал наявності будь-якої активної аварії візка
      qw_Alarm_Word : Word;   // Повна декомпозиція аварій для діагностики HMI
      qw_Status_Word : Word;   // Розширене слово стану візка (7 станів)
   END_VAR
   VAR
      EmerBrake_TON : TON_TIME;   // Таймер накладання аварійного гальма (1 хв)
      BrakeTimeout_TON : TON_TIME;   // Таймер контролю часу розгальмування
      MotionActive : Bool;   // Ознака активного запиту на рух
      stat_ZeroBlockActive : Bool;   // Прапорець активації нульового захисту
      stat_OldGlobalAlarm : Bool;   // Пам'ять попереднього стану аварії для логіки фронтів
      statAlarmWord : Word;   // Статичне слово збереження аварій
   END_VAR
   VAR_TEMP
      GlobalBlock : Bool;   // Загальна заборона руху візка
      Block_Forward : Bool;   // Блокування руху Вперед
      Block_Backward : Bool;   // Блокування руху Назад
      Valid_Cmd_Fwd : Bool;   // Валідована команда Вперед
      Valid_Cmd_Bwd : Bool;   // Валідована команда Назад
      tempStatusWord : Word;   // Тимчасова змінна для збірки слова стану
      AtForwardLimit : Bool;   // Прапорець крайнього положення Вперед
      AtBackwardLimit : Bool;   // Прапорець крайнього положення Назад
      ResetTrigger : Bool;   // Фронт скидання аварії
   END_VAR
BEGIN

       // 1. ФОРМУВАННЯ ТА ФІКСАЦІЯ АВАРІЙ У СЛОВІ (LATCH LOGIC)
       // Bit 0: Аварійний стоп крана
       IF #ix_EmergencyStop THEN
           #statAlarmWord.%X0 := TRUE;
       END_IF;

       // Bit 1: Головний контактор вимкнений під час роботи
       IF NOT #ix_MainContactorON AND (#is_RemCtrl.Btn_Fwd OR #is_RemCtrl.Btn_Bwd OR #qx_Drive_Enable) THEN
           #statAlarmWord.%X1 := TRUE;
       END_IF;

       // Bit 2: Перегрів гальмівного резистора візка (2BT1)
       IF NOT #ix_2BT1_ThermalResistor THEN
           #statAlarmWord.%X2 := TRUE;
       END_IF;

       // Bit 3: Перегрів двигуна візка (2KT)
       IF NOT #ix_2KT_ThermalMotor THEN
           #statAlarmWord.%X3 := TRUE;
       END_IF;

       // Bit 4: Несправність частотного перетворювача 2UZ1 по мережі Profinet
       IF #ix_Fault_3UZ1 THEN
           #statAlarmWord.%X4 := TRUE;
       END_IF;

       // Bit 5: Аварія при зникненні сигналу готовності енкодера (Encoder_RDY = FALSE)
       IF NOT #ix_Encoder_RDY THEN
           #statAlarmWord.%X5 := TRUE;
       END_IF;

       // Bit 6: Перевищення номінального вантажу крана 115% (ОВП)
       IF NOT #ix_1K11_Overload115 THEN
           #statAlarmWord.%X6 := TRUE;
       END_IF;

       // Пам'ять загальної аварії перед квітуванням
       #stat_OldGlobalAlarm := #statAlarmWord <> 16#0000;

       // 2. СКИДАННЯ АВАРІЙНИХ БІТІВ (КВІТУВАННЯ)
       IF #ix_Cmd_ResetAlarm THEN
           IF NOT #ix_EmergencyStop THEN
               #statAlarmWord.%X0 := FALSE;
           END_IF;
           IF #ix_MainContactorON THEN
               #statAlarmWord.%X1 := FALSE;
           END_IF;
           IF #ix_2BT1_ThermalResistor THEN
               #statAlarmWord.%X2 := FALSE;
           END_IF;
           IF  #ix_2KT_ThermalMotor THEN
               #statAlarmWord.%X3 := FALSE;
           END_IF;
           IF NOT #ix_Fault_3UZ1 THEN
               #statAlarmWord.%X4 := FALSE;
           END_IF;
           IF #ix_1K11_Overload115 THEN
               #statAlarmWord.%X6 := FALSE;
           END_IF;
       END_IF;
           // Аварія енкодера очиститься тільки якщо він фізично знову ГОТОВИЙ (Encoder_RDY = TRUE)
           IF #ix_Encoder_RDY THEN
               #statAlarmWord.%X5 := FALSE;
           END_IF;



       #qw_Alarm_Word := #statAlarmWord;
       #qx_Global_Alarm := #statAlarmWord <> 16#0000;

       // 3. КОНТРОЛЬ НУЛЬОВИХ БЛОКУВАНЬ (ЗАХИСТ ВІД ЗАКЛИНЮВАННЯ КНОПОК / ДЖОЙСТИКА)
       #ResetTrigger := #stat_OldGlobalAlarm AND NOT #qx_Global_Alarm;

       IF #ResetTrigger AND (#is_RemCtrl.Btn_Fwd OR #is_RemCtrl.Btn_Bwd) THEN
           #stat_ZeroBlockActive := TRUE;
       END_IF;

       IF NOT #is_RemCtrl.Btn_Fwd AND NOT #is_RemCtrl.Btn_Bwd THEN
           #stat_ZeroBlockActive := FALSE;
       END_IF;

       // 4. ЗАГАЛЬНА ЗАБОРОНА РУХУ
       //New Code 2026-08-11 - O.Husiev
       #GlobalBlock :=
       #qx_Global_Alarm
       OR NOT #ix_MainContactorON
       OR #stat_ZeroBlockActive
       OR (NOT #ix_Calibrated AND NOT #ix_CalibrationActive);


       // 5. ОКРЕМІ ТЕХНОЛОГІЧНІ БЛОКУВАННЯ НАПРЯМКІВ
       //New Code 2026-08-11 - O.Husiev
       #Block_Forward :=
       NOT #is_MovePerm.Forward
       OR #ix_Zone_ProgStopFwd
       OR #ix_CalibrationBlockForward;

       #Block_Backward :=
       NOT #is_MovePerm.Backward
       OR #ix_Zone_ProgStopBwd
       OR #ix_CalibrationBlockBackward
       OR ((NOT #is_MovePerm.No_Pillar) AND ((NOT #is_SpeedPerm.Speed_normal_Bwd)OR #ix_Zone_BackPreStop) AND #is_RemCtrl.Btn_Bwd);

       // 6. ВАЛІДАЦІЯ КОМАНД ТА ДОЗВІЛ ХОДУ
       #Valid_Cmd_Fwd := #is_RemCtrl.Btn_Fwd AND NOT #GlobalBlock AND NOT #Block_Forward;
       #Valid_Cmd_Bwd := #is_RemCtrl.Btn_Bwd AND NOT #GlobalBlock AND NOT #Block_Backward;

       // 7. СВІТЛОВА СИГНАЛІЗАЦІЯ ГОТОВНОСТІ ВІЗКА (2HL)
       #qx_2HL_Ready := NOT #GlobalBlock AND #ix_Calibrated AND #is_MovePerm.Forward AND #is_MovePerm.Backward;

       // 8. К КЕРУВАННЯ РУЧНИМ ГАЛЬМОМ ВІЗКА (2MB1 -> 2KM1)
       IF #ix_DriveReleaseBrakeCmd AND NOT #GlobalBlock THEN
           #qx_2KM1_WorkingBrake := TRUE;  // Розгальмувати
       ELSE
           #qx_2KM1_WorkingBrake := FALSE; // Накласти гальмо
       END_IF;

       // 9. К КЕРУВАННЯ ЧП ВІЗКА ЧЕРЕЗ PROFINET
       #qx_Drive_Enable := #Valid_Cmd_Fwd OR #Valid_Cmd_Bwd;
       //#qx_Drive_QuickStop := (#is_RemCtrl.Btn_Fwd AND #ix_Zone_ProgStopFwd) OR (#is_RemCtrl.Btn_Bwd AND #ix_Zone_ProgStopBwd) OR #statAlarmWord.%X4;
       //New Code 2026-08-11 O.Husiev
       #qx_Drive_QuickStop :=
       (#is_RemCtrl.Btn_Fwd AND #ix_Zone_ProgStopFwd)
       OR (#is_RemCtrl.Btn_Bwd AND #ix_Zone_ProgStopBwd)
       OR #statAlarmWord.%X4
       OR #ix_CalibrationQuickStop;


       // ЛОГІКА РЕГУЛЮВАННЯ ШВИДКОСТІ (+ Вперед, - Назад)
       IF NOT #qx_Drive_Enable THEN
           #qr_Drive_SpeedSetpoint := 0.0;
       ELSIF #Valid_Cmd_Fwd THEN
           //New Code 2026-08-11 O.Husiev
           IF #is_RemCtrl.Btn_ScndSpeed
               AND #is_SpeedPerm.Speed_normal_Fwd
               AND NOT #ix_CalibrationActive
           THEN

               #qr_Drive_SpeedSetpoint := 1500.0;

           ELSE

               #qr_Drive_SpeedSetpoint := 150.0;

           END_IF;

       ELSIF #Valid_Cmd_Bwd THEN
             //New Code 2026-08-11 O.Husiev
           IF #is_RemCtrl.Btn_ScndSpeed
               AND #is_SpeedPerm.Speed_normal_Bwd
               AND NOT #ix_CalibrationActive
           THEN

               #qr_Drive_SpeedSetpoint := -1500.0;

           ELSE

               #qr_Drive_SpeedSetpoint := -150.0;

           END_IF;

       END_IF;

       // 10. ФОРМУВАННЯ СЛОВА СТАНУ ВІЗКА (Status_Word — 7 взаємовиключних станів)
       #tempStatusWord := 16#0000;

       #AtForwardLimit := (NOT #is_MovePerm.Forward) OR #ix_Zone_ProgStopFwd;
       #AtBackwardLimit := (NOT #is_MovePerm.Backward) OR #ix_Zone_ProgStopBwd;

       IF #qx_Drive_Enable AND (#qr_Drive_SpeedSetpoint > 0.0) THEN
           #tempStatusWord.%X0 := TRUE;   // Рухається вперед
       ELSIF #qx_Drive_Enable AND (#qr_Drive_SpeedSetpoint < 0.0) THEN
           #tempStatusWord.%X1 := TRUE;   // Рухається назад
       ELSE
           IF #qx_Global_Alarm THEN
               #tempStatusWord.%X4 := TRUE;   // Аварія візка
           ELSIF #stat_ZeroBlockActive THEN
               #tempStatusWord.%X3 := TRUE;   // Зупинено і НЕ готовий до роботи (активний нульовий захист)
           ELSIF #AtForwardLimit THEN
               #tempStatusWord.%X5 := TRUE;   // Зупинено у крайньому положенні Вперед
           ELSIF #AtBackwardLimit THEN
               #tempStatusWord.%X6 := TRUE;   // Зупинено у крайньому положенні Назад
           ELSIF #qx_2HL_Ready THEN
               #tempStatusWord.%X2 := TRUE;   // Зупинено і Готовий до роботи
           ELSE
               #tempStatusWord.%X3 := TRUE;   // Зупинено і НЕ готовий до роботи
           END_IF;
       END_IF;

       IF #qx_Global_Alarm THEN
           #tempStatusWord.%X4 := TRUE;
       END_IF;

       #qw_Status_Word := #tempStatusWord;
END_FUNCTION_BLOCK

FUNCTION_BLOCK "FB_Trolley_Messages"   // FB421, LAD
{ S7_Optimized_Access := 'TRUE' }
VERSION : 0.1
   VAR
      ssfbHMI_w1 : "FB_DigIn_16_XOR";
      ssfbHMI_w2 : "FB_DigIn_16_XOR";
      ssfbHMI_w3 : "FB_DigIn_16_XOR";
      sarrxhmf : Array[0..10] of Bool;
   END_VAR
   VAR_TEMP
      txStartMovement : Bool;   // Початок руху механізма
      txStopMovement : Bool;   // Кінець руху механізма
      twTemp : Word;
   END_VAR
   VAR_TEMP   // added for the SCL form of the ladder/FBD networks
      _w1 : Bool;
      _w2 : Bool;
      _w3 : Bool;
      _w4 : Bool;
   END_VAR
BEGIN

REGION Network 1: Ініціалізація
END_REGION

REGION Network 2 (SCL)
   // початок руху
   #twTemp := "HMI_DB".Trolley_movement_mechanism.TM_Status AND W#16#3;
   #txStartMovement := #twTemp <> 0;
   // кінець руху
   #twTemp := "HMI_DB".Trolley_movement_mechanism.TM_Status AND W#2#01101100;
   #txStopMovement := #twTemp <> 0;
END_REGION

REGION Network 3: Перше слово повідомлень
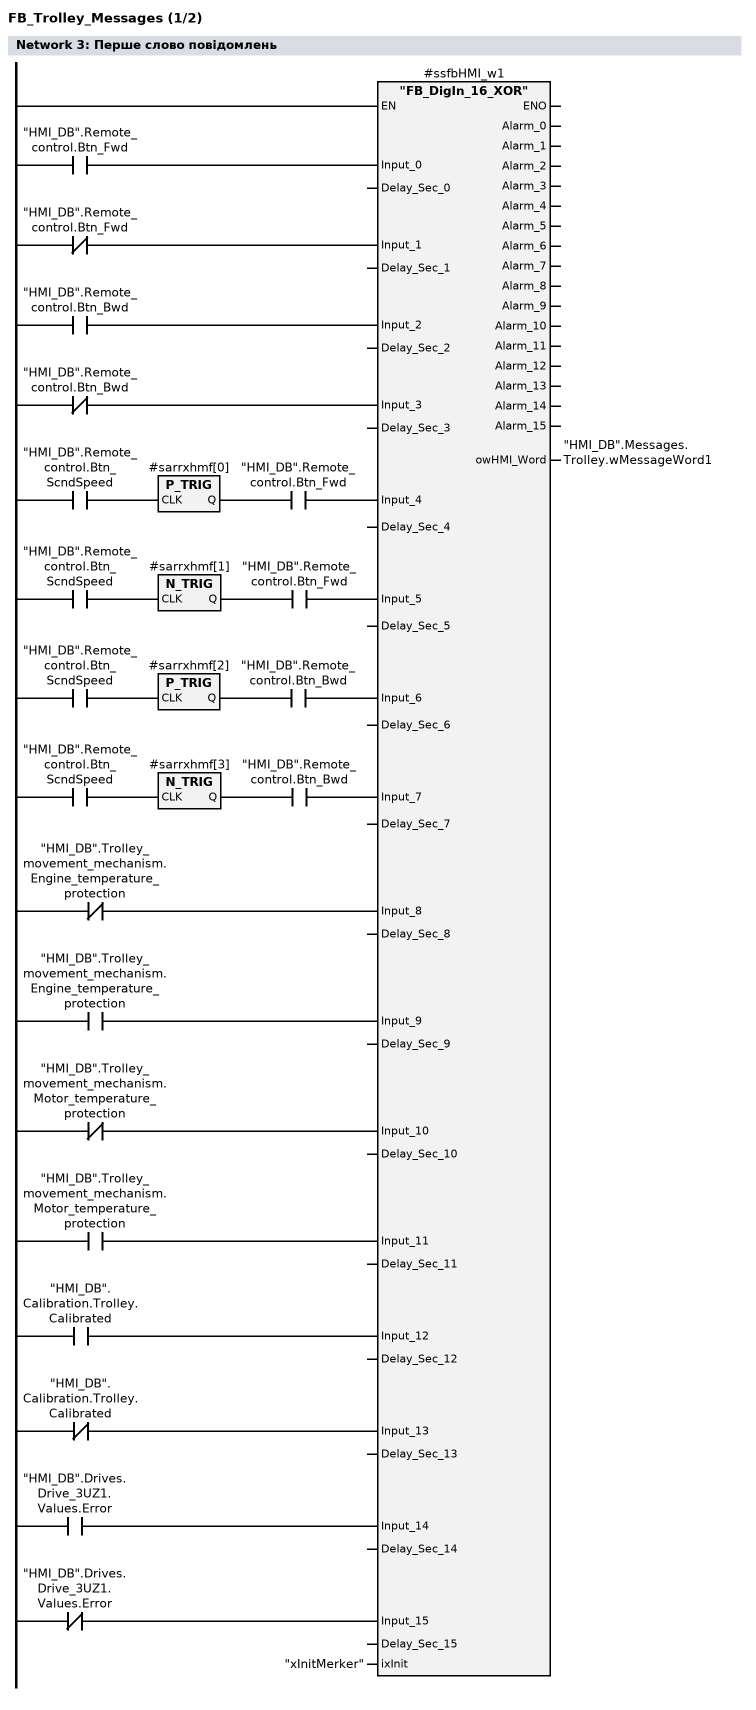
   RUNG wire#powerrail
      #ssfbHMI_w1(Input_0 := wire#w1, Input_1 := wire#w2, Input_2 := wire#w3, Input_3 := wire#w4, Input_4 := wire#w5, Input_5 := wire#w6, Input_6 := wire#w7, Input_7 := wire#w8, Input_8 := wire#w9, Input_9 := wire#w10, Input_10 := wire#w11, Input_11 := wire#w12, Input_12 := wire#w13, Input_13 := wire#w14, Input_14 := wire#w15, Input_15 := wire#w16, Delay_Sec_0 :=, Delay_Sec_1 :=, Delay_Sec_2 :=, Delay_Sec_3 :=, Delay_Sec_4 :=, Delay_Sec_5 :=, Delay_Sec_6 :=, Delay_Sec_7 :=, Delay_Sec_8 :=, Delay_Sec_9 :=, Delay_Sec_10 :=, Delay_Sec_11 :=, Delay_Sec_12 :=, Delay_Sec_13 :=, Delay_Sec_14 :=, Delay_Sec_15 :=, ixInit := "xInitMerker", Alarm_0 =>, Alarm_1 =>, Alarm_2 =>, Alarm_3 =>, Alarm_4 =>, Alarm_5 =>, Alarm_6 =>, Alarm_7 =>, Alarm_8 =>, Alarm_9 =>, Alarm_10 =>, Alarm_11 =>, Alarm_12 =>, Alarm_13 =>, Alarm_14 =>, Alarm_15 =>, owHMI_Word => "HMI_DB".Messages.Trolley.wMessageWord1)
   END_RUNG
   RUNG wire#powerrail
      Contact( "HMI_DB".Remote_control.Btn_Fwd )
   END_RUNG wire#w1
   RUNG wire#powerrail
      I_Contact( "HMI_DB".Remote_control.Btn_Fwd )
   END_RUNG wire#w2
   RUNG wire#powerrail
      Contact( "HMI_DB".Remote_control.Btn_Bwd )
   END_RUNG wire#w3
   RUNG wire#powerrail
      I_Contact( "HMI_DB".Remote_control.Btn_Bwd )
   END_RUNG wire#w4
   RUNG wire#powerrail
      Contact( "HMI_DB".Remote_control.Btn_ScndSpeed )
      P_Trig( #sarrxhmf[0] )
      Contact( "HMI_DB".Remote_control.Btn_Fwd )
   END_RUNG wire#w5
   RUNG wire#powerrail
      Contact( "HMI_DB".Remote_control.Btn_ScndSpeed )
      N_Trig( #sarrxhmf[1] )
      Contact( "HMI_DB".Remote_control.Btn_Fwd )
   END_RUNG wire#w6
   RUNG wire#powerrail
      Contact( "HMI_DB".Remote_control.Btn_ScndSpeed )
      P_Trig( #sarrxhmf[2] )
      Contact( "HMI_DB".Remote_control.Btn_Bwd )
   END_RUNG wire#w7
   RUNG wire#powerrail
      Contact( "HMI_DB".Remote_control.Btn_ScndSpeed )
      N_Trig( #sarrxhmf[3] )
      Contact( "HMI_DB".Remote_control.Btn_Bwd )
   END_RUNG wire#w8
   RUNG wire#powerrail
      I_Contact( "HMI_DB".Trolley_movement_mechanism.Engine_temperature_protection )
   END_RUNG wire#w9
   RUNG wire#powerrail
      Contact( "HMI_DB".Trolley_movement_mechanism.Engine_temperature_protection )
   END_RUNG wire#w10
   RUNG wire#powerrail
      I_Contact( "HMI_DB".Trolley_movement_mechanism.Motor_temperature_protection )
   END_RUNG wire#w11
   RUNG wire#powerrail
      Contact( "HMI_DB".Trolley_movement_mechanism.Motor_temperature_protection )
   END_RUNG wire#w12
   RUNG wire#powerrail
      Contact( "HMI_DB".Calibration.Trolley.Calibrated )
   END_RUNG wire#w13
   RUNG wire#powerrail
      I_Contact( "HMI_DB".Calibration.Trolley.Calibrated )
   END_RUNG wire#w14
   RUNG wire#powerrail
      Contact( "HMI_DB".Drives.Drive_3UZ1.Values.Error )
   END_RUNG wire#w15
   RUNG wire#powerrail
      I_Contact( "HMI_DB".Drives.Drive_3UZ1.Values.Error )
   END_RUNG wire#w16
   // the same network as SCL:
   #_w1 := "HMI_DB".Remote_control.Btn_ScndSpeed AND NOT #sarrxhmf[0];   // rising edge
   #sarrxhmf[0] := "HMI_DB".Remote_control.Btn_ScndSpeed;
   #_w2 := NOT "HMI_DB".Remote_control.Btn_ScndSpeed AND #sarrxhmf[1];   // falling edge
   #sarrxhmf[1] := "HMI_DB".Remote_control.Btn_ScndSpeed;
   #_w3 := "HMI_DB".Remote_control.Btn_ScndSpeed AND NOT #sarrxhmf[2];   // rising edge
   #sarrxhmf[2] := "HMI_DB".Remote_control.Btn_ScndSpeed;
   #_w4 := NOT "HMI_DB".Remote_control.Btn_ScndSpeed AND #sarrxhmf[3];   // falling edge
   #sarrxhmf[3] := "HMI_DB".Remote_control.Btn_ScndSpeed;
   #ssfbHMI_w1(Input_0 := "HMI_DB".Remote_control.Btn_Fwd,   // "FB_DigIn_16_XOR"
               Input_1 := NOT "HMI_DB".Remote_control.Btn_Fwd,
               Input_2 := "HMI_DB".Remote_control.Btn_Bwd,
               Input_3 := NOT "HMI_DB".Remote_control.Btn_Bwd,
               Input_4 := #_w1 AND "HMI_DB".Remote_control.Btn_Fwd,
               Input_5 := #_w2 AND "HMI_DB".Remote_control.Btn_Fwd,
               Input_6 := #_w3 AND "HMI_DB".Remote_control.Btn_Bwd,
               Input_7 := #_w4 AND "HMI_DB".Remote_control.Btn_Bwd,
               Input_8 := NOT "HMI_DB".Trolley_movement_mechanism.Engine_temperature_protection,
               Input_9 := "HMI_DB".Trolley_movement_mechanism.Engine_temperature_protection,
               Input_10 := NOT "HMI_DB".Trolley_movement_mechanism.Motor_temperature_protection,
               Input_11 := "HMI_DB".Trolley_movement_mechanism.Motor_temperature_protection,
               Input_12 := "HMI_DB".Calibration.Trolley.Calibrated,
               Input_13 := NOT "HMI_DB".Calibration.Trolley.Calibrated,
               Input_14 := "HMI_DB".Drives.Drive_3UZ1.Values.Error,
               Input_15 := NOT "HMI_DB".Drives.Drive_3UZ1.Values.Error,
               ixInit := "xInitMerker",
               owHMI_Word => "HMI_DB".Messages.Trolley.wMessageWord1);
END_REGION

REGION Network 4: Друге слово повідомлень
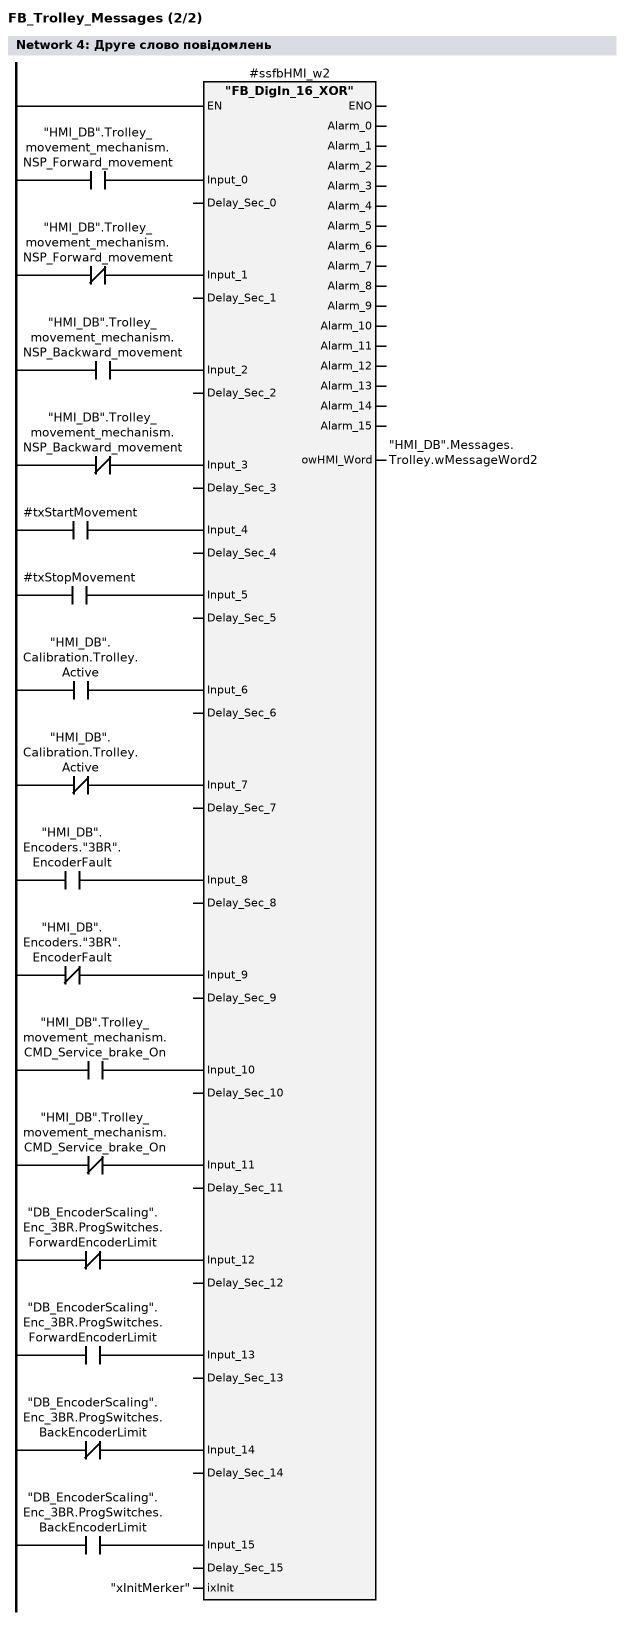
   RUNG wire#powerrail
      #ssfbHMI_w2(Input_0 := wire#w1, Input_1 := wire#w2, Input_2 := wire#w3, Input_3 := wire#w4, Input_4 := wire#w5, Input_5 := wire#w6, Input_6 := wire#w7, Input_7 := wire#w8, Input_8 := wire#w9, Input_9 := wire#w10, Input_10 := wire#w11, Input_11 := wire#w12, Input_12 := wire#w13, Input_13 := wire#w14, Input_14 := wire#w15, Input_15 := wire#w16, Delay_Sec_0 :=, Delay_Sec_1 :=, Delay_Sec_2 :=, Delay_Sec_3 :=, Delay_Sec_4 :=, Delay_Sec_5 :=, Delay_Sec_6 :=, Delay_Sec_7 :=, Delay_Sec_8 :=, Delay_Sec_9 :=, Delay_Sec_10 :=, Delay_Sec_11 :=, Delay_Sec_12 :=, Delay_Sec_13 :=, Delay_Sec_14 :=, Delay_Sec_15 :=, ixInit := "xInitMerker", Alarm_0 =>, Alarm_1 =>, Alarm_2 =>, Alarm_3 =>, Alarm_4 =>, Alarm_5 =>, Alarm_6 =>, Alarm_7 =>, Alarm_8 =>, Alarm_9 =>, Alarm_10 =>, Alarm_11 =>, Alarm_12 =>, Alarm_13 =>, Alarm_14 =>, Alarm_15 =>, owHMI_Word => "HMI_DB".Messages.Trolley.wMessageWord2)
   END_RUNG
   RUNG wire#powerrail
      Contact( "HMI_DB".Trolley_movement_mechanism.NSP_Forward_movement )
   END_RUNG wire#w1
   RUNG wire#powerrail
      I_Contact( "HMI_DB".Trolley_movement_mechanism.NSP_Forward_movement )
   END_RUNG wire#w2
   RUNG wire#powerrail
      Contact( "HMI_DB".Trolley_movement_mechanism.NSP_Backward_movement )
   END_RUNG wire#w3
   RUNG wire#powerrail
      I_Contact( "HMI_DB".Trolley_movement_mechanism.NSP_Backward_movement )
   END_RUNG wire#w4
   RUNG wire#powerrail
      Contact( #txStartMovement )
   END_RUNG wire#w5
   RUNG wire#powerrail
      Contact( #txStopMovement )
   END_RUNG wire#w6
   RUNG wire#powerrail
      Contact( "HMI_DB".Calibration.Trolley.Active )
   END_RUNG wire#w7
   RUNG wire#powerrail
      I_Contact( "HMI_DB".Calibration.Trolley.Active )
   END_RUNG wire#w8
   RUNG wire#powerrail
      Contact( "HMI_DB".Encoders."3BR".EncoderFault )
   END_RUNG wire#w9
   RUNG wire#powerrail
      I_Contact( "HMI_DB".Encoders."3BR".EncoderFault )
   END_RUNG wire#w10
   RUNG wire#powerrail
      Contact( "HMI_DB".Trolley_movement_mechanism.CMD_Service_brake_On )
   END_RUNG wire#w11
   RUNG wire#powerrail
      I_Contact( "HMI_DB".Trolley_movement_mechanism.CMD_Service_brake_On )
   END_RUNG wire#w12
   RUNG wire#powerrail
      I_Contact( "DB_EncoderScaling".Enc_3BR.ProgSwitches.ForwardEncoderLimit )
   END_RUNG wire#w13
   RUNG wire#powerrail
      Contact( "DB_EncoderScaling".Enc_3BR.ProgSwitches.ForwardEncoderLimit )
   END_RUNG wire#w14
   RUNG wire#powerrail
      I_Contact( "DB_EncoderScaling".Enc_3BR.ProgSwitches.BackEncoderLimit )
   END_RUNG wire#w15
   RUNG wire#powerrail
      Contact( "DB_EncoderScaling".Enc_3BR.ProgSwitches.BackEncoderLimit )
   END_RUNG wire#w16
   // the same network as SCL:
   #ssfbHMI_w2(Input_0 := "HMI_DB".Trolley_movement_mechanism.NSP_Forward_movement,   // "FB_DigIn_16_XOR"
               Input_1 := NOT "HMI_DB".Trolley_movement_mechanism.NSP_Forward_movement,
               Input_2 := "HMI_DB".Trolley_movement_mechanism.NSP_Backward_movement,
               Input_3 := NOT "HMI_DB".Trolley_movement_mechanism.NSP_Backward_movement,
               Input_4 := #txStartMovement,
               Input_5 := #txStopMovement,
               Input_6 := "HMI_DB".Calibration.Trolley.Active,
               Input_7 := NOT "HMI_DB".Calibration.Trolley.Active,
               Input_8 := "HMI_DB".Encoders."3BR".EncoderFault,
               Input_9 := NOT "HMI_DB".Encoders."3BR".EncoderFault,
               Input_10 := "HMI_DB".Trolley_movement_mechanism.CMD_Service_brake_On,
               Input_11 := NOT "HMI_DB".Trolley_movement_mechanism.CMD_Service_brake_On,
               Input_12 := NOT "DB_EncoderScaling".Enc_3BR.ProgSwitches.ForwardEncoderLimit,
               Input_13 := "DB_EncoderScaling".Enc_3BR.ProgSwitches.ForwardEncoderLimit,
               Input_14 := NOT "DB_EncoderScaling".Enc_3BR.ProgSwitches.BackEncoderLimit,
               Input_15 := "DB_EncoderScaling".Enc_3BR.ProgSwitches.BackEncoderLimit,
               ixInit := "xInitMerker",
               owHMI_Word => "HMI_DB".Messages.Trolley.wMessageWord2);
END_REGION
END_FUNCTION_BLOCK

FUNCTION "FC_Trolley_movement" : Void   // FC400, LAD
{ S7_Optimized_Access := 'TRUE' }
VERSION : 0.1
   VAR_TEMP   // added for the SCL form of the ladder/FBD networks
      _w1 : Bool;
   END_VAR
BEGIN

REGION Network 2: =================Блокування пристрою ручного керування========================
END_REGION

REGION Network 3: Механізм пересування візка. Дозвіл роботи (РП роз'єднан з приводом)
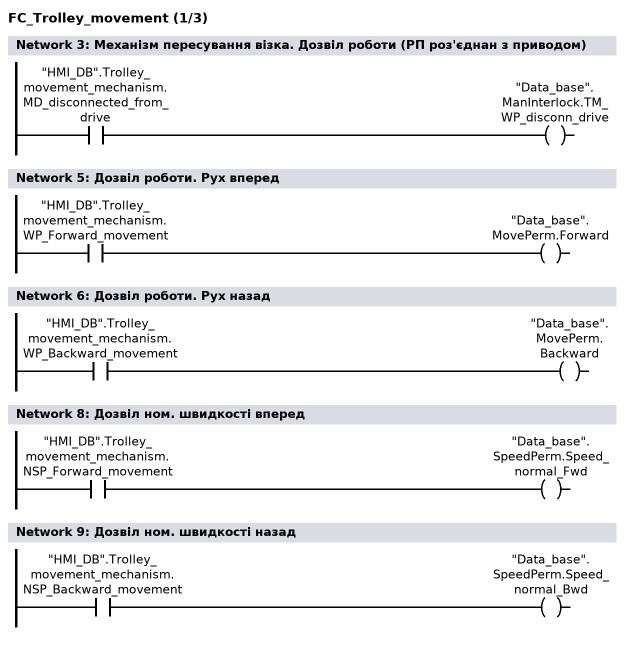
   RUNG wire#powerrail
      Contact( "HMI_DB".Trolley_movement_mechanism.MD_disconnected_from_drive )
      Coil( "Data_base".ManInterlock.TM_WP_disconn_drive )
   END_RUNG
   // the same network as SCL:
   "Data_base".ManInterlock.TM_WP_disconn_drive := "HMI_DB".Trolley_movement_mechanism.MD_disconnected_from_drive;
END_REGION

REGION Network 4: ================Дозвіл роботи====================
END_REGION

REGION Network 5: Дозвіл роботи. Рух вперед
   RUNG wire#powerrail
      Contact( "HMI_DB".Trolley_movement_mechanism.WP_Forward_movement )
      Coil( "Data_base".MovePerm.Forward )
   END_RUNG
   // the same network as SCL:
   "Data_base".MovePerm.Forward := "HMI_DB".Trolley_movement_mechanism.WP_Forward_movement;
END_REGION

REGION Network 6: Дозвіл роботи. Рух назад
   RUNG wire#powerrail
      Contact( "HMI_DB".Trolley_movement_mechanism.WP_Backward_movement )
      Coil( "Data_base".MovePerm.Backward )
   END_RUNG
   // the same network as SCL:
   "Data_base".MovePerm.Backward := "HMI_DB".Trolley_movement_mechanism.WP_Backward_movement;
END_REGION

REGION Network 7: ================Дозвіл нормальної швидкості =================
END_REGION

REGION Network 8: Дозвіл ном. швидкості вперед
   RUNG wire#powerrail
      Contact( "HMI_DB".Trolley_movement_mechanism.NSP_Forward_movement )
      Coil( "Data_base".SpeedPerm.Speed_normal_Fwd )
   END_RUNG
   // the same network as SCL:
   "Data_base".SpeedPerm.Speed_normal_Fwd := "HMI_DB".Trolley_movement_mechanism.NSP_Forward_movement;
END_REGION

REGION Network 9: Дозвіл ном. швидкості назад
   RUNG wire#powerrail
      Contact( "HMI_DB".Trolley_movement_mechanism.NSP_Backward_movement )
      Coil( "Data_base".SpeedPerm.Speed_normal_Bwd )
   END_RUNG
   // the same network as SCL:
   "Data_base".SpeedPerm.Speed_normal_Bwd := "HMI_DB".Trolley_movement_mechanism.NSP_Backward_movement;
END_REGION

REGION Network 10: ===============Керування механізмом візка================ / ===============Керування механізмом підйому================
END_REGION

REGION Network 11: Механізм візка
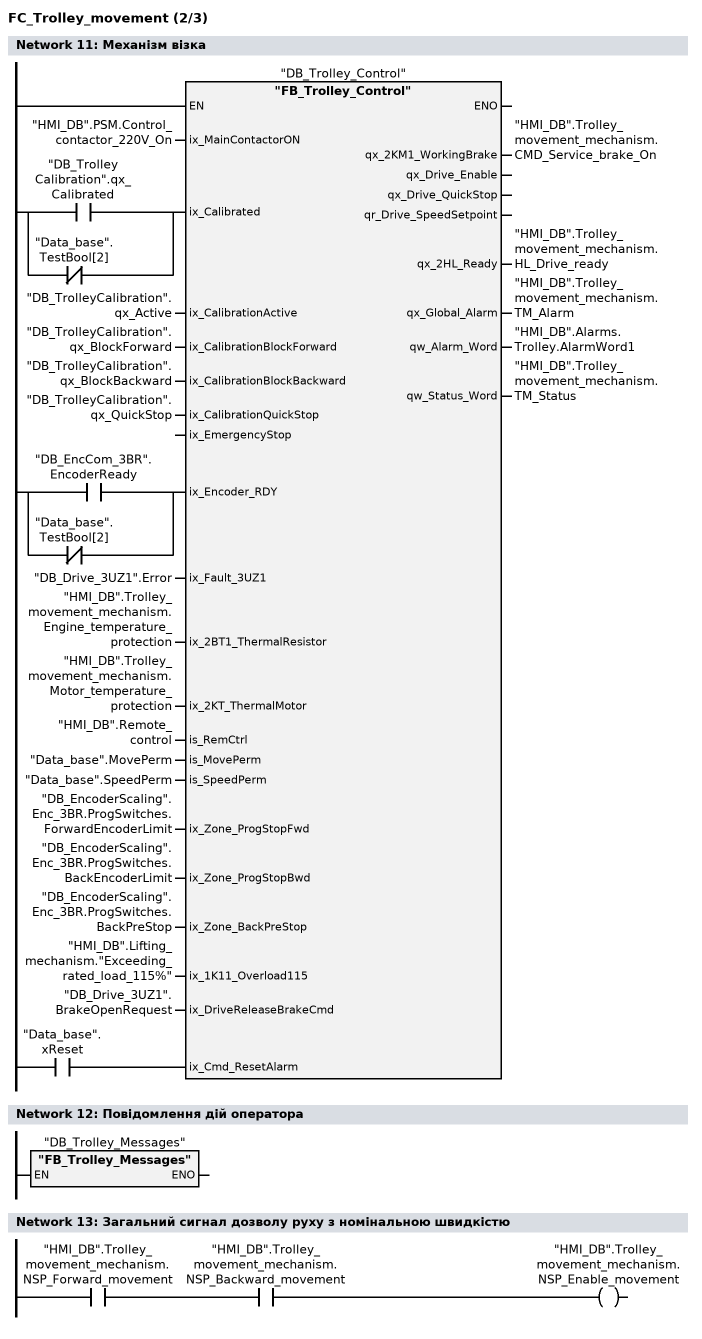
   RUNG wire#powerrail
      "DB_Trolley_Control"(ix_Calibrated := wire#w1, ix_Encoder_RDY := wire#w2, ix_Cmd_ResetAlarm := wire#w3, ix_MainContactorON := "HMI_DB".PSM.Control_contactor_220V_On, ix_CalibrationActive := "DB_TrolleyCalibration".qx_Active, ix_CalibrationBlockForward := "DB_TrolleyCalibration".qx_BlockForward, ix_CalibrationBlockBackward := "DB_TrolleyCalibration".qx_BlockBackward, ix_CalibrationQuickStop := "DB_TrolleyCalibration".qx_QuickStop, ix_EmergencyStop :=, ix_Fault_3UZ1 := "DB_Drive_3UZ1".Error, ix_2BT1_ThermalResistor := "HMI_DB".Trolley_movement_mechanism.Engine_temperature_protection, ix_2KT_ThermalMotor := "HMI_DB".Trolley_movement_mechanism.Motor_temperature_protection, is_RemCtrl := "HMI_DB".Remote_control, is_MovePerm := "Data_base".MovePerm, is_SpeedPerm := "Data_base".SpeedPerm, ix_Zone_ProgStopFwd := "DB_EncoderScaling".Enc_3BR.ProgSwitches.ForwardEncoderLimit, ix_Zone_ProgStopBwd := "DB_EncoderScaling".Enc_3BR.ProgSwitches.BackEncoderLimit, ix_Zone_BackPreStop := "DB_EncoderScaling".Enc_3BR.ProgSwitches.BackPreStop, ix_1K11_Overload115 := "HMI_DB".Lifting_mechanism."Exceeding_rated_load_115%", ix_DriveReleaseBrakeCmd := "DB_Drive_3UZ1".BrakeOpenRequest, qx_2KM1_WorkingBrake => "HMI_DB".Trolley_movement_mechanism.CMD_Service_brake_On, qx_Drive_Enable =>, qx_Drive_QuickStop =>, qr_Drive_SpeedSetpoint =>, qx_2HL_Ready => "HMI_DB".Trolley_movement_mechanism.HL_Drive_ready, qx_Global_Alarm => "HMI_DB".Trolley_movement_mechanism.TM_Alarm, qw_Alarm_Word => "HMI_DB".Alarms.Trolley.AlarmWord1, qw_Status_Word => "HMI_DB".Trolley_movement_mechanism.TM_Status)
   END_RUNG
   RUNG wire#powerrail
      Contact( "DB_TrolleyCalibration".qx_Calibrated )
   END_RUNG wire#w1
   RUNG wire#powerrail
      I_Contact( "Data_base".TestBool[2] )
   END_RUNG wire#w1
   RUNG wire#powerrail
      Contact( "DB_EncCom_3BR".EncoderReady )
   END_RUNG wire#w2
   RUNG wire#powerrail
      I_Contact( "Data_base".TestBool[2] )
   END_RUNG wire#w2
   RUNG wire#powerrail
      Contact( "Data_base".xReset )
   END_RUNG wire#w3
   // the same network as SCL:
   "DB_Trolley_Control"(ix_MainContactorON := "HMI_DB".PSM.Control_contactor_220V_On,   // "FB_Trolley_Control"
                        ix_Calibrated := "DB_TrolleyCalibration".qx_Calibrated OR NOT "Data_base".TestBool[2],
                        ix_CalibrationActive := "DB_TrolleyCalibration".qx_Active,
                        ix_CalibrationBlockForward := "DB_TrolleyCalibration".qx_BlockForward,
                        ix_CalibrationBlockBackward := "DB_TrolleyCalibration".qx_BlockBackward,
                        ix_CalibrationQuickStop := "DB_TrolleyCalibration".qx_QuickStop,
                        ix_Encoder_RDY := "DB_EncCom_3BR".EncoderReady OR NOT "Data_base".TestBool[2],
                        ix_Fault_3UZ1 := "DB_Drive_3UZ1".Error,
                        ix_2BT1_ThermalResistor := "HMI_DB".Trolley_movement_mechanism.Engine_temperature_protection,
                        ix_2KT_ThermalMotor := "HMI_DB".Trolley_movement_mechanism.Motor_temperature_protection,
                        is_RemCtrl := "HMI_DB".Remote_control,
                        is_MovePerm := "Data_base".MovePerm,
                        is_SpeedPerm := "Data_base".SpeedPerm,
                        ix_Zone_ProgStopFwd := "DB_EncoderScaling".Enc_3BR.ProgSwitches.ForwardEncoderLimit,
                        ix_Zone_ProgStopBwd := "DB_EncoderScaling".Enc_3BR.ProgSwitches.BackEncoderLimit,
                        ix_Zone_BackPreStop := "DB_EncoderScaling".Enc_3BR.ProgSwitches.BackPreStop,
                        ix_1K11_Overload115 := "HMI_DB".Lifting_mechanism."Exceeding_rated_load_115%",
                        ix_DriveReleaseBrakeCmd := "DB_Drive_3UZ1".BrakeOpenRequest,
                        ix_Cmd_ResetAlarm := "Data_base".xReset,
                        qx_2KM1_WorkingBrake => "HMI_DB".Trolley_movement_mechanism.CMD_Service_brake_On,
                        qx_2HL_Ready => "HMI_DB".Trolley_movement_mechanism.HL_Drive_ready,
                        qx_Global_Alarm => "HMI_DB".Trolley_movement_mechanism.TM_Alarm,
                        qw_Alarm_Word => "HMI_DB".Alarms.Trolley.AlarmWord1,
                        qw_Status_Word => "HMI_DB".Trolley_movement_mechanism.TM_Status);
END_REGION

REGION Network 12: Повідомлення дій оператора
   RUNG wire#powerrail
      "DB_Trolley_Messages"()
   END_RUNG
   // the same network as SCL:
   "DB_Trolley_Messages"();   // "FB_Trolley_Messages"
END_REGION

REGION Network 13: Загальний сигнал дозволу руху з номінальною швидкістю
   RUNG wire#powerrail
      Contact( "HMI_DB".Trolley_movement_mechanism.NSP_Forward_movement )
      Contact( "HMI_DB".Trolley_movement_mechanism.NSP_Backward_movement )
      Coil( "HMI_DB".Trolley_movement_mechanism.NSP_Enable_movement )
   END_RUNG
   // the same network as SCL:
   "HMI_DB".Trolley_movement_mechanism.NSP_Enable_movement := "HMI_DB".Trolley_movement_mechanism.NSP_Forward_movement AND "HMI_DB".Trolley_movement_mechanism.NSP_Backward_movement;
END_REGION

REGION Network 14: Рух з другою та першою швидкістю команда
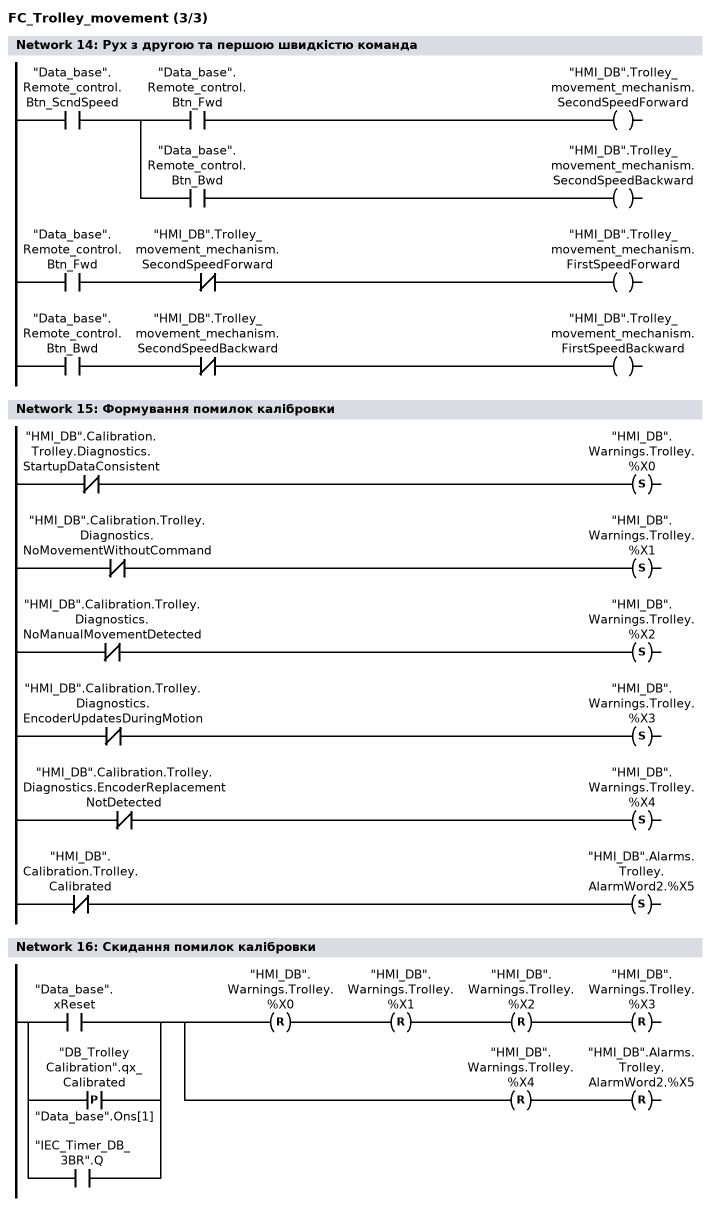
   RUNG wire#powerrail
      Contact( "Data_base".Remote_control.Btn_ScndSpeed )
      wire#w1
      Contact( "Data_base".Remote_control.Btn_Fwd )
      Coil( "HMI_DB".Trolley_movement_mechanism.SecondSpeedForward )
   END_RUNG
   RUNG wire#w1
      Contact( "Data_base".Remote_control.Btn_Bwd )
      Coil( "HMI_DB".Trolley_movement_mechanism.SecondSpeedBackward )
   END_RUNG
   RUNG wire#powerrail
      Contact( "Data_base".Remote_control.Btn_Fwd )
      I_Contact( "HMI_DB".Trolley_movement_mechanism.SecondSpeedForward )
      Coil( "HMI_DB".Trolley_movement_mechanism.FirstSpeedForward )
   END_RUNG
   RUNG wire#powerrail
      Contact( "Data_base".Remote_control.Btn_Bwd )
      I_Contact( "HMI_DB".Trolley_movement_mechanism.SecondSpeedBackward )
      Coil( "HMI_DB".Trolley_movement_mechanism.FirstSpeedBackward )
   END_RUNG
   // the same network as SCL:
   "HMI_DB".Trolley_movement_mechanism.SecondSpeedForward := "Data_base".Remote_control.Btn_ScndSpeed AND "Data_base".Remote_control.Btn_Fwd;
   "HMI_DB".Trolley_movement_mechanism.SecondSpeedBackward := "Data_base".Remote_control.Btn_ScndSpeed AND "Data_base".Remote_control.Btn_Bwd;
   "HMI_DB".Trolley_movement_mechanism.FirstSpeedForward := "Data_base".Remote_control.Btn_Fwd AND NOT "HMI_DB".Trolley_movement_mechanism.SecondSpeedForward;
   "HMI_DB".Trolley_movement_mechanism.FirstSpeedBackward := "Data_base".Remote_control.Btn_Bwd AND NOT "HMI_DB".Trolley_movement_mechanism.SecondSpeedBackward;
END_REGION

REGION Network 15: Формування помилок калібровки
   RUNG wire#powerrail
      I_Contact( "HMI_DB".Calibration.Trolley.Diagnostics.StartupDataConsistent )
      S_Coil( "HMI_DB".Warnings.Trolley.%X0 )
   END_RUNG
   RUNG wire#powerrail
      I_Contact( "HMI_DB".Calibration.Trolley.Diagnostics.NoMovementWithoutCommand )
      S_Coil( "HMI_DB".Warnings.Trolley.%X1 )
   END_RUNG
   RUNG wire#powerrail
      I_Contact( "HMI_DB".Calibration.Trolley.Diagnostics.NoManualMovementDetected )
      S_Coil( "HMI_DB".Warnings.Trolley.%X2 )
   END_RUNG
   RUNG wire#powerrail
      I_Contact( "HMI_DB".Calibration.Trolley.Diagnostics.EncoderUpdatesDuringMotion )
      S_Coil( "HMI_DB".Warnings.Trolley.%X3 )
   END_RUNG
   RUNG wire#powerrail
      I_Contact( "HMI_DB".Calibration.Trolley.Diagnostics.EncoderReplacementNotDetected )
      S_Coil( "HMI_DB".Warnings.Trolley.%X4 )
   END_RUNG
   RUNG wire#powerrail
      I_Contact( "HMI_DB".Calibration.Trolley.Calibrated )
      S_Coil( "HMI_DB".Alarms.Trolley.AlarmWord2.%X5 )
   END_RUNG
   // the same network as SCL:
   IF NOT "HMI_DB".Calibration.Trolley.Diagnostics.StartupDataConsistent THEN
       "HMI_DB".Warnings.Trolley.%X0 := TRUE;
   END_IF;
   IF NOT "HMI_DB".Calibration.Trolley.Diagnostics.NoMovementWithoutCommand THEN
       "HMI_DB".Warnings.Trolley.%X1 := TRUE;
   END_IF;
   IF NOT "HMI_DB".Calibration.Trolley.Diagnostics.NoManualMovementDetected THEN
       "HMI_DB".Warnings.Trolley.%X2 := TRUE;
   END_IF;
   IF NOT "HMI_DB".Calibration.Trolley.Diagnostics.EncoderUpdatesDuringMotion THEN
       "HMI_DB".Warnings.Trolley.%X3 := TRUE;
   END_IF;
   IF NOT "HMI_DB".Calibration.Trolley.Diagnostics.EncoderReplacementNotDetected THEN
       "HMI_DB".Warnings.Trolley.%X4 := TRUE;
   END_IF;
   IF NOT "HMI_DB".Calibration.Trolley.Calibrated THEN
       "HMI_DB".Alarms.Trolley.AlarmWord2.%X5 := TRUE;
   END_IF;
END_REGION

REGION Network 16: Скидання помилок калібровки
   RUNG wire#powerrail
      Contact( "Data_base".xReset )
      wire#w1
      R_Coil( "HMI_DB".Warnings.Trolley.%X0 )
      R_Coil( "HMI_DB".Warnings.Trolley.%X1 )
      R_Coil( "HMI_DB".Warnings.Trolley.%X2 )
      R_Coil( "HMI_DB".Warnings.Trolley.%X3 )
   END_RUNG
   RUNG wire#powerrail
      P_Contact(operand := "DB_TrolleyCalibration".qx_Calibrated, bit := "Data_base".Ons[1])
   END_RUNG wire#w1
   RUNG wire#powerrail
      Contact( "IEC_Timer_DB_3BR".Q )
   END_RUNG wire#w1
   RUNG wire#w1
      R_Coil( "HMI_DB".Warnings.Trolley.%X4 )
      R_Coil( "HMI_DB".Alarms.Trolley.AlarmWord2.%X5 )
   END_RUNG
   // the same network as SCL:
   #_w1 := "DB_TrolleyCalibration".qx_Calibrated AND NOT "Data_base".Ons[1];   // rising edge of "DB_TrolleyCalibration".qx_Calibrated
   "Data_base".Ons[1] := "DB_TrolleyCalibration".qx_Calibrated;
   IF "Data_base".xReset OR #_w1 OR "IEC_Timer_DB_3BR".Q THEN
       "HMI_DB".Warnings.Trolley.%X0 := FALSE;
       "HMI_DB".Warnings.Trolley.%X1 := FALSE;
       "HMI_DB".Warnings.Trolley.%X2 := FALSE;
       "HMI_DB".Warnings.Trolley.%X3 := FALSE;
       "HMI_DB".Warnings.Trolley.%X4 := FALSE;
       "HMI_DB".Alarms.Trolley.AlarmWord2.%X5 := FALSE;
   END_IF;
END_REGION
END_FUNCTION

// folder: 5000_Setup

FUNCTION "FC_Setup" : Void   // FC5001, SCL
{ S7_Optimized_Access := 'TRUE' }
VERSION : 0.1
BEGIN

   //Механізм підйому. Вимикачі кінцеві на гальмі 1YB2. Гальмо розгальмоване
   //"HMI_DB".IO_Tags.OutCfg.DigOut_0_2.SML := 1;
   //"HMI_DB".IO_Tags.OutCfg.DigOut_0_2.SVal := 1;
   //"HMI_DB".IO_Tags.InCnf.DigIn_5_3.SML := 1;
   //"HMI_DB".IO_Tags.InCnf.DigIn_5_3.SVal := 1;

   //Контроль обертання барабану
   //"HMI_DB".IO_Tags.InCnf.DigIn_3_1.SML := 1;
   //"HMI_DB".IO_Tags.InCnf.DigIn_3_1.SVal := 1;

   //invertion rotation encoder
   "Data_base".TestReal[0] := "DB_Lifting_Control".qr_Drive_SpeedSetpoint * (1);
END_FUNCTION

// folder: 500_4UZ1_4UZ2_Crane_movement(CM)

FUNCTION_BLOCK "FB_Crane_Control"   // FB500, SCL
{ S7_Optimized_Access := 'TRUE' }
VERSION : 0.1
   VAR_INPUT
      ix_MainContactorON : Bool;   // Головний контактор увімкнено
      ix_Calibrated : Bool;   // Механізм моста калібровано по енкодерах
      ix_CalibrationActive : Bool;   // Активна процедура калібровки моста
      ix_CalibrationBlockForward : Bool;   // Заборона руху вперед / вправо від блока калібровки
      ix_CalibrationBlockBackward : Bool;   // Заборона руху назад / вліво від блока калібровки
      ix_CalibrationQuickStop : Bool;   // Запит Quick Stop від блока калібровки
      ix_EmergencyStop : Bool;   // Загальний аварійний стоп
      ix_Encoder1_RDY : Bool;   // Готовність енкодера 1
      ix_Encoder2_RDY : Bool;   // Готовність енкодера 2
      ix_Fault_4UZ1 : Bool;   // Аварія лівого ЧП 4UZ1
      ix_Fault_4UZ2 : Bool;   // Аварія лівого ЧП 4UZ2
      ix_4BT1_ThermalResistor : Bool;   // Термостат гальмівного резистора лівого приводу
      ix_4BT2_ThermalResistor : Bool;   // Термостат гальмівного резистора правого приводу
      ix_4KT1_ThermalMotor : Bool;   // Термісторне реле двигуна лівого приводу 4M1
      ix_4KT2_ThermalMotor : Bool;   // Термісторне реле двигуна правого приводу 4M2
      ir_4UZ1_Actual_Speed : Real;   // Фактична швидкість лівого приводу 4UZ1 (об/хв)
      ir_4UZ2_Actual_Speed : Real;   // Фактична швидкість правого приводу 4UZ2 (об/хв)
      id_Pos_Encoder1_MM : DInt;   // Поточне положення лівої опори (4UZ1) в мм
      id_Pos_Encoder2_MM : DInt;   // Поточне положення правої опори (4UZ2) в мм
      id_Max_Skew_Limit_MM : DInt := 50;   // Уставка максимального перекосу в мм (дефолт 50 мм)
      is_RemCtrl : "udtRemCtrl";   // Кнопки руху з пульта (для контролю нульового положення при старті)
      is_MovePerm : "udtMovePerm";   // Кінцеві вимикачі руху крайніх положень
      is_SpeedPerm : "udtSpeedPerm";   // Кінцеві вимикачі швидкості руху
      ix_Zone_ProgStopFwd : Bool;   // Програмна зона зупинки Вперед/Вліво
      ix_Zone_ProgStopBwd : Bool;   // Програмна зона зупинки Назад/Вправо
      ix_PilarZoneLimit : Bool;   // Дозвіл роботи. Збудь-якої зі сторін від колони
      ix_1K11_Overload115 : Bool;   // Відсутність сигналу = Перевантаження 115%
      ix_Drive1ReleaseBrakeCmd : Bool;   // Команда розгальмування від ЧП 4UZ1 в телеграмі
      ix_Drive2ReleaseBrakeCmd : Bool;   // Команда розгальмування від ЧП 4UZ2 в телеграмі
      ix_Cmd_ResetAlarm : Bool;   // Кнопка скидання аварій (квітування)
   END_VAR
   VAR_OUTPUT
      qx_4KM1_WorkingBrake : Bool;   // Пускач зовнішнього робочого гальма
      qx_Drive_Enable : Bool;   // Загальний сигнал дозволу руху для обох ЧП
      qx_Drive_QuickStop : Bool;   // Команда швидкого гальмування Quick Stop (OFF3) для обох ЧП
      qr_Drive_SpeedSetpoint : Real;   // Завдання швидкості на ЧП зі знаком (- Вперед/Вліво, + Назад/Вправо)
      qx_4HL_Ready : Bool;   // Світловий індикатор готовності моста
      qx_Global_Alarm : Bool;   // Сигнал наявності будь-якої активної аварії моста
      qw_Alarm_Word : Word;   // Повна декомпозиція аварій для діагностики HMI
      qw_Status_Word : Word;   // Розширене слово стану моста (7 станів)
   END_VAR
   VAR
      statAlarmWord : Word;   // Статичне слово збереження аварій
      stat_ZeroBlockActive : Bool;   // Прапорець активації нульового захисту
      stat_OldGlobalAlarm : Bool;   // Пам'ять попереднього стану аварії для логіки фронтів
      stat_SetRightBlock : Bool;
      stat_SetLeftBlock : Bool;
      T_SpeedDiffDelay : TON_TIME;
   END_VAR
   VAR_TEMP
      GlobalBlock : Bool;
      Block_Forward : Bool;
      Block_Backward : Bool;
      Valid_Cmd_Fwd : Bool;
      Valid_Cmd_Bwd : Bool;
      AtForwardLimit : Bool;
      AtBackwardLimit : Bool;
      ResetTrigger : Bool;
      tempStatusWord : Word;
      Current_Skew_MM : DInt;
      SpeedDiff : Bool;
      SpeedDiffDelayTime : DInt;
   END_VAR
BEGIN

       // 1. ФОРМУВАННЯ ТА ФІКСАЦІЯ АВАРІЙ У СЛОВІ (LATCH LOGIC)
       // Bit 0: Аварійний стоп крана
       IF #ix_EmergencyStop THEN
           #statAlarmWord.%X0 := TRUE;
       END_IF;

       // Bit 1: Головний контактор вимкнений під час роботи
       IF NOT #ix_MainContactorON AND (#is_RemCtrl.Btn_Right OR #is_RemCtrl.Btn_Left OR #qx_Drive_Enable) THEN
           #statAlarmWord.%X1 := TRUE;
       END_IF;

       // Bit 2: Перегрів гальмівного резистора 4BT1
       IF NOT #ix_4BT1_ThermalResistor THEN
           #statAlarmWord.%X2 := TRUE;
       END_IF;

       // Bit 3: Перегрів гальмівного резистора 4BT2
       IF NOT #ix_4BT2_ThermalResistor THEN
           #statAlarmWord.%X3 := TRUE;
       END_IF;

       // Bit 4: Перегрів лівого двигуна моста за сигналами термісторного реле 4KT1
       IF NOT #ix_4KT1_ThermalMotor THEN
           #statAlarmWord.%X4 := TRUE;
       END_IF;

       // Bit 5: Перегрів лівого двигуна моста за сигналами термісторного реле 4KT2
       IF NOT #ix_4KT2_ThermalMotor THEN
           #statAlarmWord.%X5 := TRUE;
       END_IF;

       // Bit 6: Внутрішня несправність частотних перетворювачів 4UZ1
       IF #ix_Fault_4UZ1 THEN
           #statAlarmWord.%X6 := TRUE;
       END_IF;

       // Bit 7: Внутрішня несправність частотних перетворювачів 4UZ2
       IF #ix_Fault_4UZ2 THEN
           #statAlarmWord.%X7 := TRUE;
       END_IF;

       // Bit 8: Втрата готовності енкодера Encoder1
       IF NOT #ix_Encoder1_RDY THEN
           #statAlarmWord.%X8 := TRUE;
       END_IF;

       // Bit 9: Втрата готовності енкодера Encoder2
       IF NOT #ix_Encoder2_RDY THEN
           #statAlarmWord.%X9 := TRUE;
       END_IF;

       // Bit 10: Перевищення номінального вантажу крана 115% (ОВП)
       IF NOT #ix_1K11_Overload115 THEN
           #statAlarmWord.%X10 := TRUE;
       END_IF;

       // Bit 11: Динамічний перекіс по швидкості двигунів (Розбіжність > 150 об/хв під час ходу)

       IF #qx_Drive_Enable AND (ABS(#"ir_4UZ1_Actual_Speed" - #"ir_4UZ2_Actual_Speed") > 150.0) THEN
           #SpeedDiff := TRUE;
       END_IF;

       #T_SpeedDiffDelay(IN := #SpeedDiff,
                         PT := T#2S,
                         Q => #statAlarmWord.%X11,
                         ET =>#SpeedDiffDelayTime);

       // Bit 12: НОВА АВАРІЯ — Критичний статичний перекіс моста по датчиках енкодерів у міліметрах
       // Обчислюємо абсолютну різницю між координатами лівої та правої ніг
       #Current_Skew_MM := ABS(#id_Pos_Encoder1_MM - #id_Pos_Encoder2_MM);
       // Захист активний, якщо механізм відкалібрований і перевищено виставлений ліміт уставки
       IF #ix_Calibrated AND (#Current_Skew_MM > #id_Max_Skew_Limit_MM) THEN
           #statAlarmWord.%X12 := TRUE;
       END_IF;

       // Пам'ять загальної аварії перед квітуванням
       #stat_OldGlobalAlarm := #statAlarmWord <> 16#0000;

       // 2. СКИДАННЯ АВАРІЙНИХ БІТІВ (КВІТУВАННЯ)
       IF #ix_Cmd_ResetAlarm THEN
           IF NOT #ix_EmergencyStop THEN
               #statAlarmWord.%X0 := FALSE;
           END_IF;
           IF #ix_MainContactorON THEN
               #statAlarmWord.%X1 := FALSE;
           END_IF;
           IF #ix_4BT1_ThermalResistor THEN
               #statAlarmWord.%X2 := FALSE;
           END_IF;
           IF #ix_4BT2_ThermalResistor THEN
               #statAlarmWord.%X3 := FALSE;
           END_IF;
           IF  #ix_4KT1_ThermalMotor THEN
               #statAlarmWord.%X4 := FALSE;
           END_IF;
           IF #ix_4KT2_ThermalMotor THEN
               #statAlarmWord.%X5 := FALSE;
           END_IF;
           IF NOT #ix_Fault_4UZ1 THEN
               #statAlarmWord.%X6 := FALSE;
           END_IF;
           IF NOT #ix_Fault_4UZ2 THEN
               #statAlarmWord.%X7 := FALSE;
           END_IF;
           IF #ix_Encoder1_RDY THEN
               #statAlarmWord.%X8 := FALSE;
           END_IF;
           IF #ix_Encoder2_RDY THEN
               #statAlarmWord.%X9 := FALSE;
           END_IF;
           IF #ix_1K11_Overload115 THEN
               #statAlarmWord.%X10 := FALSE;
           END_IF;

           #statAlarmWord.%X11 := FALSE; // Скидання динамічного перекосу

           // Аварія перекосу в мм очиститься тільки якщо геометрична різниця стала меншою за уставку
           IF #Current_Skew_MM <= #id_Max_Skew_Limit_MM THEN
               #statAlarmWord.%X12 := FALSE;
           END_IF;
       END_IF;

       #qw_Alarm_Word := #statAlarmWord;
       #qx_Global_Alarm := #statAlarmWord <> 16#0000;

       // 3. КОНТРОЛЬ НУЛЬОВИХ БЛОКУВАНЬ
       #ResetTrigger := #stat_OldGlobalAlarm AND NOT #qx_Global_Alarm;

       IF #ResetTrigger AND (#is_RemCtrl.Btn_Right OR #is_RemCtrl.Btn_Left) THEN
           #stat_ZeroBlockActive := TRUE;
       END_IF;

       IF NOT #is_RemCtrl.Btn_Right AND NOT #is_RemCtrl.Btn_Left THEN
           #stat_ZeroBlockActive := FALSE;
       END_IF;

       // 4. ЗАГАЛЬНА ЗАБОРОНА РУХУ
       //New Code 2026-08-12 O.Husiev
       #GlobalBlock :=
       #qx_Global_Alarm
       OR NOT #ix_MainContactorON
       OR #stat_ZeroBlockActive
       OR (NOT #ix_Calibrated AND NOT #ix_CalibrationActive);

       // 5. ОКРЕМІ ТЕХНОЛОГІЧНІ БЛОКУВАННЯ НАПРЯМКІВ
       // New Code 2026-08-15 DZH 
       IF  (NOT #is_MovePerm.No_Pillar OR NOT #ix_PilarZoneLimit) AND  NOT #is_SpeedPerm.Speed_normal_Bwd AND
           #is_RemCtrl.Btn_Right AND NOT #stat_SetLeftBlock THEN
           #stat_SetRightBlock:=true;
       END_IF;
       IF (#is_MovePerm.No_Pillar AND #ix_PilarZoneLimit) OR #is_SpeedPerm.Speed_normal_Bwd THEN
           #stat_SetRightBlock:=FALSE;
       END_IF;

       IF (NOT #is_MovePerm.No_Pillar OR NOT #ix_PilarZoneLimit) AND NOT #is_SpeedPerm.Speed_normal_Bwd AND
           #is_RemCtrl.Btn_Left AND NOT #stat_SetRightBlock THEN
           #stat_SetLeftBlock:= TRUE ;
       END_IF;
       IF (#is_MovePerm.No_Pillar AND #ix_PilarZoneLimit) OR #is_SpeedPerm.Speed_normal_Bwd  THEN
           #stat_SetLeftBlock := FALSE;
       END_IF;


       //New Code 2026-08-12 O.Husiev
       #Block_Forward :=
       NOT #is_MovePerm.Right
       OR #ix_Zone_ProgStopFwd
       OR #ix_CalibrationBlockForward;
    //   OR #stat_SetRightBlock;//New Code 2026-08-15 DZH

       #Block_Backward :=
       NOT #is_MovePerm.Left
       OR #ix_Zone_ProgStopBwd
       OR #ix_CalibrationBlockBackward;
   //    OR #stat_SetLeftBlock;//New Code 2026-08-15 DZH

       // 6. ВАЛІДАЦІЯ КОМАНД ТА ДОЗВІЛ ХОДУ
       #Valid_Cmd_Fwd := #is_RemCtrl.Btn_Right AND NOT #GlobalBlock AND NOT #Block_Forward;
       #Valid_Cmd_Bwd := #is_RemCtrl.Btn_Left AND NOT #GlobalBlock AND NOT #Block_Backward;

       // 7. СВІТЛОВА СИГНАЛІЗАЦІЯ ГОТОВНОСТІ МОСТА (4HL)
       #"qx_4HL_Ready" := NOT #GlobalBlock AND #ix_Calibrated AND #is_MovePerm.Right AND #is_MovePerm.Left;

       // 8. К КЕРУВАННЯ РУЧНИМИ ГАЛЬМАМИ ОПОР МОСТА (4MB1 -> 4KM1)
       IF #ix_Drive1ReleaseBrakeCmd AND #ix_Drive2ReleaseBrakeCmd AND NOT #GlobalBlock THEN
           #"qx_4KM1_WorkingBrake" := TRUE;
       ELSE
           #"qx_4KM1_WorkingBrake" := FALSE;
       END_IF;


       // 9. К КЕРУВАННЯ ЧП МОСТА ЧЕРЕЗ PROFINET
       #qx_Drive_Enable := #Valid_Cmd_Fwd OR #Valid_Cmd_Bwd;

       //New Code 2026-08-12 - O.Husiev
       #qx_Drive_QuickStop :=
       (#is_RemCtrl.Btn_Right AND #ix_Zone_ProgStopFwd)
       OR (#is_RemCtrl.Btn_Left AND #ix_Zone_ProgStopBwd)
       OR #statAlarmWord.%X4
       OR #ix_CalibrationQuickStop;

       // ЛОГІКА РЕГУЛЮВАННЯ ШВИДКОСТІ (+ Вперед/Вліво, - Назад/Вправо)
       IF NOT #qx_Drive_Enable THEN
           #qr_Drive_SpeedSetpoint := 0.0;
       ELSIF #Valid_Cmd_Fwd THEN
           //New Code 2026-8-12 - O.Husiev
           IF #is_RemCtrl.Btn_ScndSpeed
               AND #is_SpeedPerm.Speed_normal_Right
               AND NOT #ix_CalibrationActive
           THEN

               #qr_Drive_SpeedSetpoint := 1500.0;

           ELSE

               #qr_Drive_SpeedSetpoint := 260.0;

           END_IF;

       ELSIF #Valid_Cmd_Bwd THEN
           // New Code 2026-08-26 - O.Husiev
           IF #is_RemCtrl.Btn_ScndSpeed
               AND #is_SpeedPerm.Speed_normal_Left
               AND NOT #ix_CalibrationActive
           THEN

               #qr_Drive_SpeedSetpoint := -1500.0;

           ELSE

               #qr_Drive_SpeedSetpoint := -260.0;

           END_IF;
       END_IF;

       // 10. ФОРМУВАННЯ СЛОВА СТАНУ МОСТА (#Status_Word)
       #tempStatusWord := 16#0000;

       #AtForwardLimit := (NOT #is_MovePerm.Right) OR #ix_Zone_ProgStopFwd;
       #AtBackwardLimit := (NOT #is_MovePerm.Left) OR #ix_Zone_ProgStopBwd;

       IF #qx_Drive_Enable AND (#qr_Drive_SpeedSetpoint > 0.0) THEN
           #tempStatusWord.%X1 := TRUE;   // Рухається вперед / вліво
       ELSIF #qx_Drive_Enable AND (#qr_Drive_SpeedSetpoint < 0.0) THEN
           #tempStatusWord.%X0 := TRUE;   // Рухається назад / вправо
       ELSE
           IF #qx_Global_Alarm THEN
               #tempStatusWord.%X4 := TRUE;   // Аварія моста
           ELSIF #stat_ZeroBlockActive THEN
               #tempStatusWord.%X3 := TRUE;   // Зупинено і НЕ готовий до роботи (активний нульовий захист джойстика)  
           ELSIF #AtForwardLimit THEN
               #tempStatusWord.%X5 := TRUE;   // Зупинено у крайньому положенні Вперед/Вліво
           ELSIF #AtBackwardLimit THEN
               #tempStatusWord.%X6 := TRUE;   // Зупинено у крайньому положенні Назад/Вправо  
           ELSIF #"qx_4HL_Ready" THEN
               #tempStatusWord.%X2 := TRUE;   // Зупинено і Готовий до роботи
           ELSE
               #tempStatusWord.%X3 := TRUE;   // Зупинено і НЕ готовий до роботи
           END_IF;
           END_IF;

           IF #qx_Global_Alarm THEN
               #tempStatusWord.%X4 := TRUE;END_IF;

           #qw_Status_Word := #tempStatusWord;
END_FUNCTION_BLOCK

FUNCTION_BLOCK "FB_Crane_Messages"   // FB521, LAD
{ S7_Optimized_Access := 'TRUE' }
VERSION : 0.1
   VAR
      ssfbHMI_w1 : "FB_DigIn_16_XOR";
      ssfbHMI_w2 : "FB_DigIn_16_XOR";
      ssfbHMI_w3 : "FB_DigIn_16_XOR";
      sarrxhmf : Array[0..10] of Bool;
   END_VAR
   VAR_TEMP
      txStartMovement : Bool;   // Початок руху механізма
      txStopMovement : Bool;   // Кінець руху механізма
      twTemp : Word;
   END_VAR
   VAR_TEMP   // added for the SCL form of the ladder/FBD networks
      _w1 : Bool;
      _w2 : Bool;
      _w3 : Bool;
      _w4 : Bool;
   END_VAR
BEGIN

REGION Network 2 (SCL)
   // початок руху
   #twTemp := "HMI_DB".Crane_movement_mechanism.CM_Status AND W#16#3;
   #txStartMovement := #twTemp <> 0;
   // кінець руху
   #twTemp := "HMI_DB".Crane_movement_mechanism.CM_Status AND W#2#01101100;
   #txStopMovement := #twTemp <> 0;
END_REGION

REGION Network 3: Перше слово повідомлень
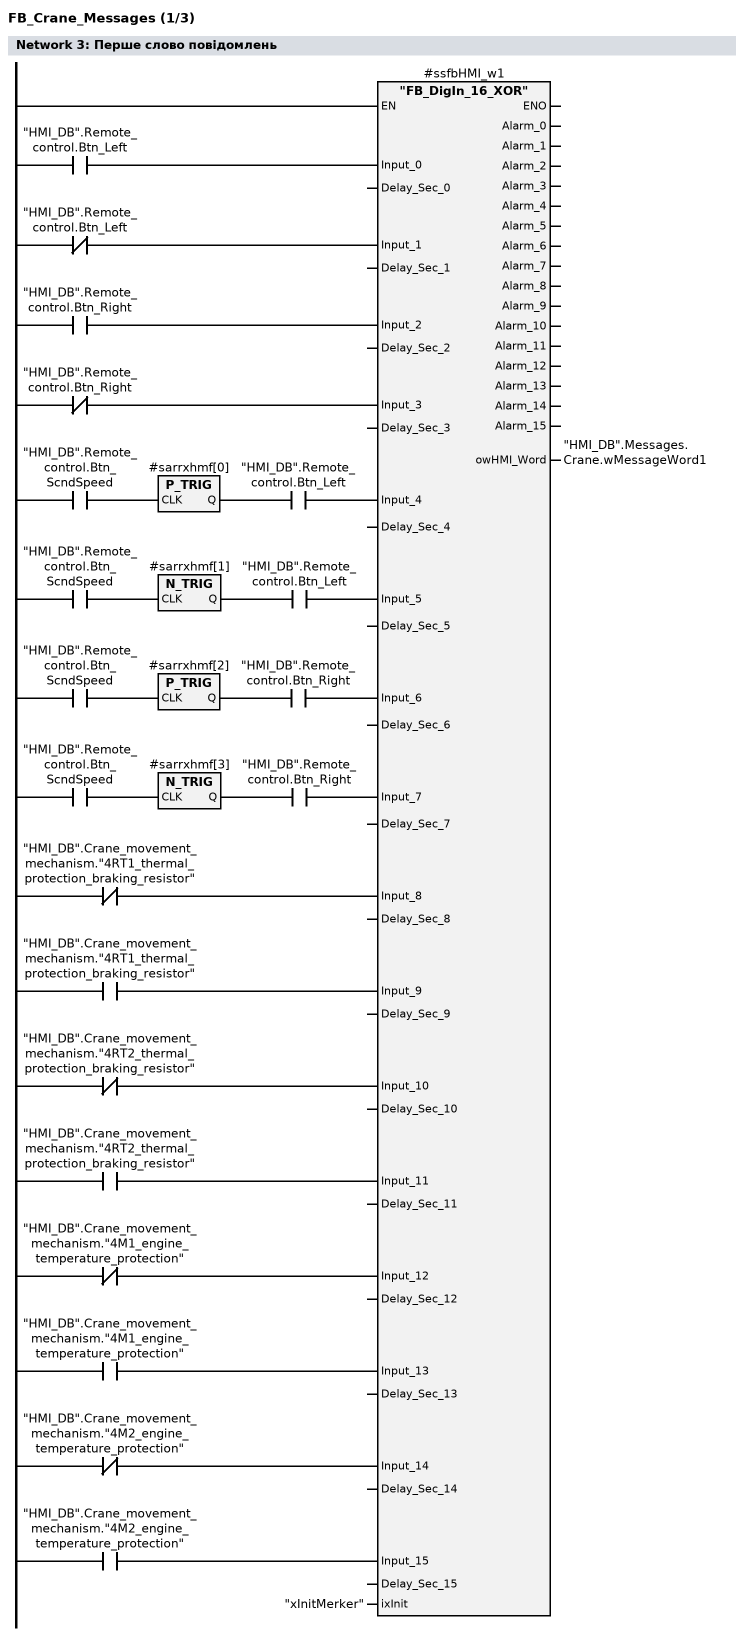
   RUNG wire#powerrail
      #ssfbHMI_w1(Input_0 := wire#w1, Input_1 := wire#w2, Input_2 := wire#w3, Input_3 := wire#w4, Input_4 := wire#w5, Input_5 := wire#w6, Input_6 := wire#w7, Input_7 := wire#w8, Input_8 := wire#w9, Input_9 := wire#w10, Input_10 := wire#w11, Input_11 := wire#w12, Input_12 := wire#w13, Input_13 := wire#w14, Input_14 := wire#w15, Input_15 := wire#w16, Delay_Sec_0 :=, Delay_Sec_1 :=, Delay_Sec_2 :=, Delay_Sec_3 :=, Delay_Sec_4 :=, Delay_Sec_5 :=, Delay_Sec_6 :=, Delay_Sec_7 :=, Delay_Sec_8 :=, Delay_Sec_9 :=, Delay_Sec_10 :=, Delay_Sec_11 :=, Delay_Sec_12 :=, Delay_Sec_13 :=, Delay_Sec_14 :=, Delay_Sec_15 :=, ixInit := "xInitMerker", Alarm_0 =>, Alarm_1 =>, Alarm_2 =>, Alarm_3 =>, Alarm_4 =>, Alarm_5 =>, Alarm_6 =>, Alarm_7 =>, Alarm_8 =>, Alarm_9 =>, Alarm_10 =>, Alarm_11 =>, Alarm_12 =>, Alarm_13 =>, Alarm_14 =>, Alarm_15 =>, owHMI_Word => "HMI_DB".Messages.Crane.wMessageWord1)
   END_RUNG
   RUNG wire#powerrail
      Contact( "HMI_DB".Remote_control.Btn_Left )
   END_RUNG wire#w1
   RUNG wire#powerrail
      I_Contact( "HMI_DB".Remote_control.Btn_Left )
   END_RUNG wire#w2
   RUNG wire#powerrail
      Contact( "HMI_DB".Remote_control.Btn_Right )
   END_RUNG wire#w3
   RUNG wire#powerrail
      I_Contact( "HMI_DB".Remote_control.Btn_Right )
   END_RUNG wire#w4
   RUNG wire#powerrail
      Contact( "HMI_DB".Remote_control.Btn_ScndSpeed )
      P_Trig( #sarrxhmf[0] )
      Contact( "HMI_DB".Remote_control.Btn_Left )
   END_RUNG wire#w5
   RUNG wire#powerrail
      Contact( "HMI_DB".Remote_control.Btn_ScndSpeed )
      N_Trig( #sarrxhmf[1] )
      Contact( "HMI_DB".Remote_control.Btn_Left )
   END_RUNG wire#w6
   RUNG wire#powerrail
      Contact( "HMI_DB".Remote_control.Btn_ScndSpeed )
      P_Trig( #sarrxhmf[2] )
      Contact( "HMI_DB".Remote_control.Btn_Right )
   END_RUNG wire#w7
   RUNG wire#powerrail
      Contact( "HMI_DB".Remote_control.Btn_ScndSpeed )
      N_Trig( #sarrxhmf[3] )
      Contact( "HMI_DB".Remote_control.Btn_Right )
   END_RUNG wire#w8
   RUNG wire#powerrail
      I_Contact( "HMI_DB".Crane_movement_mechanism."4RT1_thermal_protection_braking_resistor" )
   END_RUNG wire#w9
   RUNG wire#powerrail
      Contact( "HMI_DB".Crane_movement_mechanism."4RT1_thermal_protection_braking_resistor" )
   END_RUNG wire#w10
   RUNG wire#powerrail
      I_Contact( "HMI_DB".Crane_movement_mechanism."4RT2_thermal_protection_braking_resistor" )
   END_RUNG wire#w11
   RUNG wire#powerrail
      Contact( "HMI_DB".Crane_movement_mechanism."4RT2_thermal_protection_braking_resistor" )
   END_RUNG wire#w12
   RUNG wire#powerrail
      I_Contact( "HMI_DB".Crane_movement_mechanism."4M1_engine_temperature_protection" )
   END_RUNG wire#w13
   RUNG wire#powerrail
      Contact( "HMI_DB".Crane_movement_mechanism."4M1_engine_temperature_protection" )
   END_RUNG wire#w14
   RUNG wire#powerrail
      I_Contact( "HMI_DB".Crane_movement_mechanism."4M2_engine_temperature_protection" )
   END_RUNG wire#w15
   RUNG wire#powerrail
      Contact( "HMI_DB".Crane_movement_mechanism."4M2_engine_temperature_protection" )
   END_RUNG wire#w16
   // the same network as SCL:
   #_w1 := "HMI_DB".Remote_control.Btn_ScndSpeed AND NOT #sarrxhmf[0];   // rising edge
   #sarrxhmf[0] := "HMI_DB".Remote_control.Btn_ScndSpeed;
   #_w2 := NOT "HMI_DB".Remote_control.Btn_ScndSpeed AND #sarrxhmf[1];   // falling edge
   #sarrxhmf[1] := "HMI_DB".Remote_control.Btn_ScndSpeed;
   #_w3 := "HMI_DB".Remote_control.Btn_ScndSpeed AND NOT #sarrxhmf[2];   // rising edge
   #sarrxhmf[2] := "HMI_DB".Remote_control.Btn_ScndSpeed;
   #_w4 := NOT "HMI_DB".Remote_control.Btn_ScndSpeed AND #sarrxhmf[3];   // falling edge
   #sarrxhmf[3] := "HMI_DB".Remote_control.Btn_ScndSpeed;
   #ssfbHMI_w1(Input_0 := "HMI_DB".Remote_control.Btn_Left,   // "FB_DigIn_16_XOR"
               Input_1 := NOT "HMI_DB".Remote_control.Btn_Left,
               Input_2 := "HMI_DB".Remote_control.Btn_Right,
               Input_3 := NOT "HMI_DB".Remote_control.Btn_Right,
               Input_4 := #_w1 AND "HMI_DB".Remote_control.Btn_Left,
               Input_5 := #_w2 AND "HMI_DB".Remote_control.Btn_Left,
               Input_6 := #_w3 AND "HMI_DB".Remote_control.Btn_Right,
               Input_7 := #_w4 AND "HMI_DB".Remote_control.Btn_Right,
               Input_8 := NOT "HMI_DB".Crane_movement_mechanism."4RT1_thermal_protection_braking_resistor",
               Input_9 := "HMI_DB".Crane_movement_mechanism."4RT1_thermal_protection_braking_resistor",
               Input_10 := NOT "HMI_DB".Crane_movement_mechanism."4RT2_thermal_protection_braking_resistor",
               Input_11 := "HMI_DB".Crane_movement_mechanism."4RT2_thermal_protection_braking_resistor",
               Input_12 := NOT "HMI_DB".Crane_movement_mechanism."4M1_engine_temperature_protection",
               Input_13 := "HMI_DB".Crane_movement_mechanism."4M1_engine_temperature_protection",
               Input_14 := NOT "HMI_DB".Crane_movement_mechanism."4M2_engine_temperature_protection",
               Input_15 := "HMI_DB".Crane_movement_mechanism."4M2_engine_temperature_protection",
               ixInit := "xInitMerker",
               owHMI_Word => "HMI_DB".Messages.Crane.wMessageWord1);
END_REGION

REGION Network 4: Друге слово повідомлень
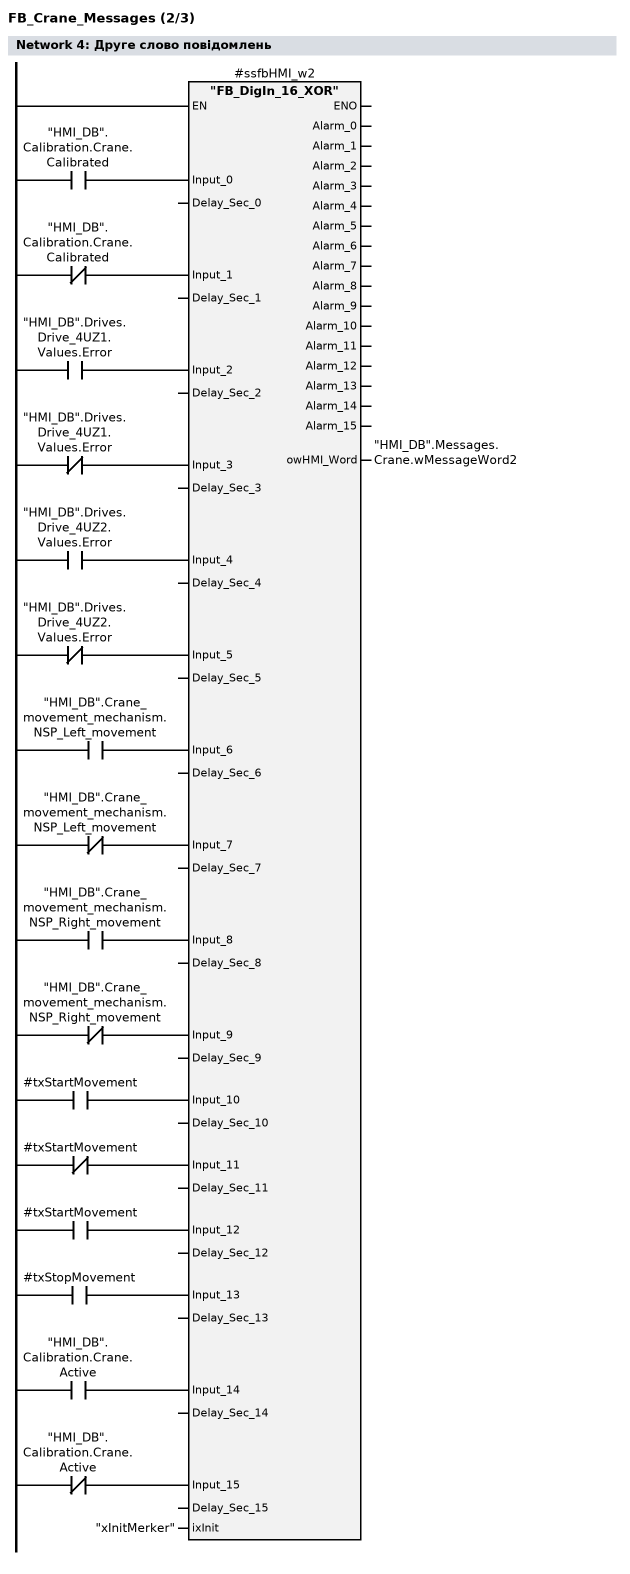
   RUNG wire#powerrail
      #ssfbHMI_w2(Input_0 := wire#w1, Input_1 := wire#w2, Input_2 := wire#w3, Input_3 := wire#w4, Input_4 := wire#w5, Input_5 := wire#w6, Input_6 := wire#w7, Input_7 := wire#w8, Input_8 := wire#w9, Input_9 := wire#w10, Input_10 := wire#w11, Input_11 := wire#w12, Input_12 := wire#w13, Input_13 := wire#w14, Input_14 := wire#w15, Input_15 := wire#w16, Delay_Sec_0 :=, Delay_Sec_1 :=, Delay_Sec_2 :=, Delay_Sec_3 :=, Delay_Sec_4 :=, Delay_Sec_5 :=, Delay_Sec_6 :=, Delay_Sec_7 :=, Delay_Sec_8 :=, Delay_Sec_9 :=, Delay_Sec_10 :=, Delay_Sec_11 :=, Delay_Sec_12 :=, Delay_Sec_13 :=, Delay_Sec_14 :=, Delay_Sec_15 :=, ixInit := "xInitMerker", Alarm_0 =>, Alarm_1 =>, Alarm_2 =>, Alarm_3 =>, Alarm_4 =>, Alarm_5 =>, Alarm_6 =>, Alarm_7 =>, Alarm_8 =>, Alarm_9 =>, Alarm_10 =>, Alarm_11 =>, Alarm_12 =>, Alarm_13 =>, Alarm_14 =>, Alarm_15 =>, owHMI_Word => "HMI_DB".Messages.Crane.wMessageWord2)
   END_RUNG
   RUNG wire#powerrail
      Contact( "HMI_DB".Calibration.Crane.Calibrated )
   END_RUNG wire#w1
   RUNG wire#powerrail
      I_Contact( "HMI_DB".Calibration.Crane.Calibrated )
   END_RUNG wire#w2
   RUNG wire#powerrail
      Contact( "HMI_DB".Drives.Drive_4UZ1.Values.Error )
   END_RUNG wire#w3
   RUNG wire#powerrail
      I_Contact( "HMI_DB".Drives.Drive_4UZ1.Values.Error )
   END_RUNG wire#w4
   RUNG wire#powerrail
      Contact( "HMI_DB".Drives.Drive_4UZ2.Values.Error )
   END_RUNG wire#w5
   RUNG wire#powerrail
      I_Contact( "HMI_DB".Drives.Drive_4UZ2.Values.Error )
   END_RUNG wire#w6
   RUNG wire#powerrail
      Contact( "HMI_DB".Crane_movement_mechanism.NSP_Left_movement )
   END_RUNG wire#w7
   RUNG wire#powerrail
      I_Contact( "HMI_DB".Crane_movement_mechanism.NSP_Left_movement )
   END_RUNG wire#w8
   RUNG wire#powerrail
      Contact( "HMI_DB".Crane_movement_mechanism.NSP_Right_movement )
   END_RUNG wire#w9
   RUNG wire#powerrail
      I_Contact( "HMI_DB".Crane_movement_mechanism.NSP_Right_movement )
   END_RUNG wire#w10
   RUNG wire#powerrail
      Contact( #txStartMovement )
   END_RUNG wire#w11
   RUNG wire#powerrail
      I_Contact( #txStartMovement )
   END_RUNG wire#w12
   RUNG wire#powerrail
      Contact( #txStartMovement )
   END_RUNG wire#w13
   RUNG wire#powerrail
      Contact( #txStopMovement )
   END_RUNG wire#w14
   RUNG wire#powerrail
      Contact( "HMI_DB".Calibration.Crane.Active )
   END_RUNG wire#w15
   RUNG wire#powerrail
      I_Contact( "HMI_DB".Calibration.Crane.Active )
   END_RUNG wire#w16
   // the same network as SCL:
   #ssfbHMI_w2(Input_0 := "HMI_DB".Calibration.Crane.Calibrated,   // "FB_DigIn_16_XOR"
               Input_1 := NOT "HMI_DB".Calibration.Crane.Calibrated,
               Input_2 := "HMI_DB".Drives.Drive_4UZ1.Values.Error,
               Input_3 := NOT "HMI_DB".Drives.Drive_4UZ1.Values.Error,
               Input_4 := "HMI_DB".Drives.Drive_4UZ2.Values.Error,
               Input_5 := NOT "HMI_DB".Drives.Drive_4UZ2.Values.Error,
               Input_6 := "HMI_DB".Crane_movement_mechanism.NSP_Left_movement,
               Input_7 := NOT "HMI_DB".Crane_movement_mechanism.NSP_Left_movement,
               Input_8 := "HMI_DB".Crane_movement_mechanism.NSP_Right_movement,
               Input_9 := NOT "HMI_DB".Crane_movement_mechanism.NSP_Right_movement,
               Input_10 := #txStartMovement,
               Input_11 := NOT #txStartMovement,
               Input_12 := #txStartMovement,
               Input_13 := #txStopMovement,
               Input_14 := "HMI_DB".Calibration.Crane.Active,
               Input_15 := NOT "HMI_DB".Calibration.Crane.Active,
               ixInit := "xInitMerker",
               owHMI_Word => "HMI_DB".Messages.Crane.wMessageWord2);
END_REGION

REGION Network 5: Третє слово повідомлень
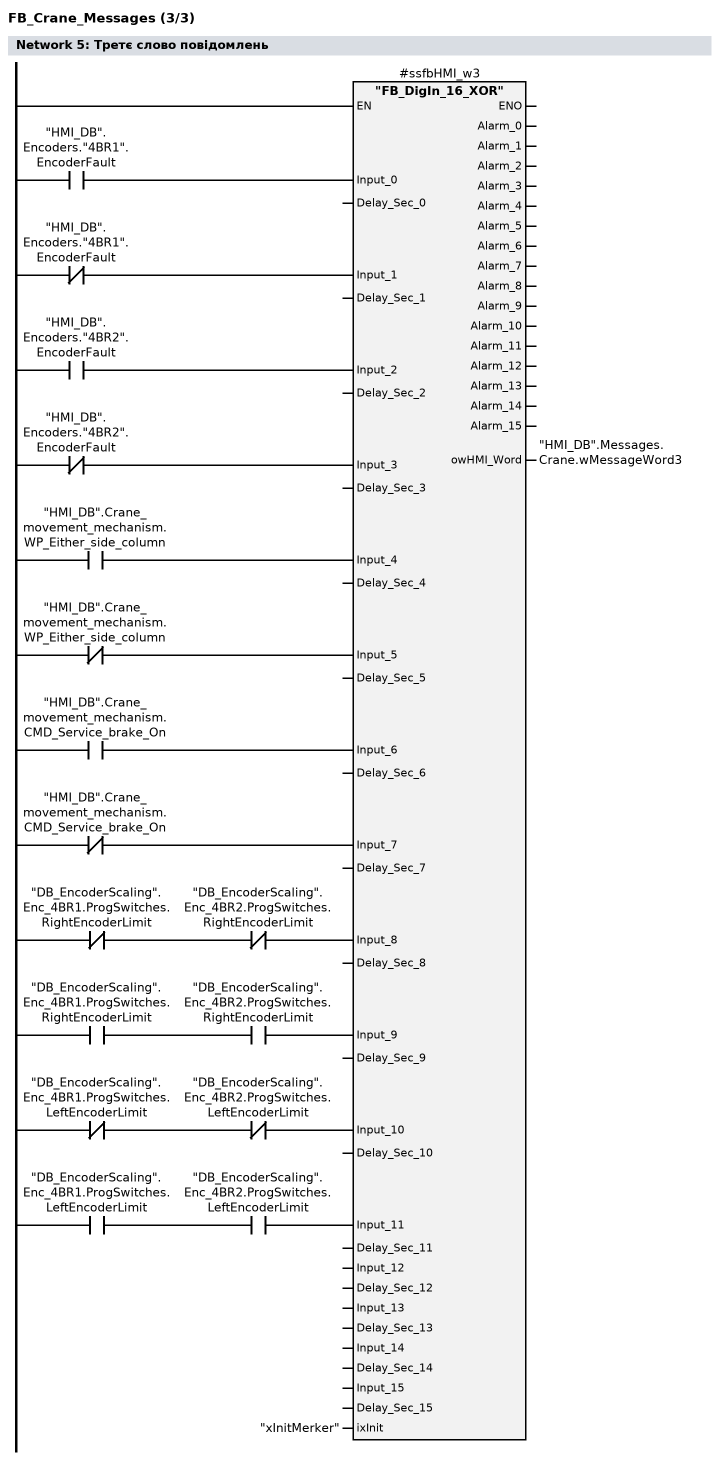
   RUNG wire#powerrail
      #ssfbHMI_w3(Input_0 := wire#w1, Input_1 := wire#w2, Input_2 := wire#w3, Input_3 := wire#w4, Input_4 := wire#w5, Input_5 := wire#w6, Input_6 := wire#w7, Input_7 := wire#w8, Input_8 := wire#w9, Input_9 := wire#w10, Input_10 := wire#w11, Input_11 := wire#w12, Delay_Sec_0 :=, Delay_Sec_1 :=, Delay_Sec_2 :=, Delay_Sec_3 :=, Delay_Sec_4 :=, Delay_Sec_5 :=, Delay_Sec_6 :=, Delay_Sec_7 :=, Delay_Sec_8 :=, Delay_Sec_9 :=, Delay_Sec_10 :=, Delay_Sec_11 :=, Input_12 :=, Delay_Sec_12 :=, Input_13 :=, Delay_Sec_13 :=, Input_14 :=, Delay_Sec_14 :=, Input_15 :=, Delay_Sec_15 :=, ixInit := "xInitMerker", Alarm_0 =>, Alarm_1 =>, Alarm_2 =>, Alarm_3 =>, Alarm_4 =>, Alarm_5 =>, Alarm_6 =>, Alarm_7 =>, Alarm_8 =>, Alarm_9 =>, Alarm_10 =>, Alarm_11 =>, Alarm_12 =>, Alarm_13 =>, Alarm_14 =>, Alarm_15 =>, owHMI_Word => "HMI_DB".Messages.Crane.wMessageWord3)
   END_RUNG
   RUNG wire#powerrail
      Contact( "HMI_DB".Encoders."4BR1".EncoderFault )
   END_RUNG wire#w1
   RUNG wire#powerrail
      I_Contact( "HMI_DB".Encoders."4BR1".EncoderFault )
   END_RUNG wire#w2
   RUNG wire#powerrail
      Contact( "HMI_DB".Encoders."4BR2".EncoderFault )
   END_RUNG wire#w3
   RUNG wire#powerrail
      I_Contact( "HMI_DB".Encoders."4BR2".EncoderFault )
   END_RUNG wire#w4
   RUNG wire#powerrail
      Contact( "HMI_DB".Crane_movement_mechanism.WP_Either_side_column )
   END_RUNG wire#w5
   RUNG wire#powerrail
      I_Contact( "HMI_DB".Crane_movement_mechanism.WP_Either_side_column )
   END_RUNG wire#w6
   RUNG wire#powerrail
      Contact( "HMI_DB".Crane_movement_mechanism.CMD_Service_brake_On )
   END_RUNG wire#w7
   RUNG wire#powerrail
      I_Contact( "HMI_DB".Crane_movement_mechanism.CMD_Service_brake_On )
   END_RUNG wire#w8
   RUNG wire#powerrail
      I_Contact( "DB_EncoderScaling".Enc_4BR1.ProgSwitches.RightEncoderLimit )
      I_Contact( "DB_EncoderScaling".Enc_4BR2.ProgSwitches.RightEncoderLimit )
   END_RUNG wire#w9
   RUNG wire#powerrail
      Contact( "DB_EncoderScaling".Enc_4BR1.ProgSwitches.RightEncoderLimit )
      Contact( "DB_EncoderScaling".Enc_4BR2.ProgSwitches.RightEncoderLimit )
   END_RUNG wire#w10
   RUNG wire#powerrail
      I_Contact( "DB_EncoderScaling".Enc_4BR1.ProgSwitches.LeftEncoderLimit )
      I_Contact( "DB_EncoderScaling".Enc_4BR2.ProgSwitches.LeftEncoderLimit )
   END_RUNG wire#w11
   RUNG wire#powerrail
      Contact( "DB_EncoderScaling".Enc_4BR1.ProgSwitches.LeftEncoderLimit )
      Contact( "DB_EncoderScaling".Enc_4BR2.ProgSwitches.LeftEncoderLimit )
   END_RUNG wire#w12
   // the same network as SCL:
   #ssfbHMI_w3(Input_0 := "HMI_DB".Encoders."4BR1".EncoderFault,   // "FB_DigIn_16_XOR"
               Input_1 := NOT "HMI_DB".Encoders."4BR1".EncoderFault,
               Input_2 := "HMI_DB".Encoders."4BR2".EncoderFault,
               Input_3 := NOT "HMI_DB".Encoders."4BR2".EncoderFault,
               Input_4 := "HMI_DB".Crane_movement_mechanism.WP_Either_side_column,
               Input_5 := NOT "HMI_DB".Crane_movement_mechanism.WP_Either_side_column,
               Input_6 := "HMI_DB".Crane_movement_mechanism.CMD_Service_brake_On,
               Input_7 := NOT "HMI_DB".Crane_movement_mechanism.CMD_Service_brake_On,
               Input_8 := NOT "DB_EncoderScaling".Enc_4BR1.ProgSwitches.RightEncoderLimit AND NOT "DB_EncoderScaling".Enc_4BR2.ProgSwitches.RightEncoderLimit,
               Input_9 := "DB_EncoderScaling".Enc_4BR1.ProgSwitches.RightEncoderLimit AND "DB_EncoderScaling".Enc_4BR2.ProgSwitches.RightEncoderLimit,
               Input_10 := NOT "DB_EncoderScaling".Enc_4BR1.ProgSwitches.LeftEncoderLimit AND NOT "DB_EncoderScaling".Enc_4BR2.ProgSwitches.LeftEncoderLimit,
               Input_11 := "DB_EncoderScaling".Enc_4BR1.ProgSwitches.LeftEncoderLimit AND "DB_EncoderScaling".Enc_4BR2.ProgSwitches.LeftEncoderLimit,
               ixInit := "xInitMerker",
               owHMI_Word => "HMI_DB".Messages.Crane.wMessageWord3);
END_REGION
END_FUNCTION_BLOCK

FUNCTION "FC_Crane_movement" : Void   // FC500, LAD
{ S7_Optimized_Access := 'TRUE' }
VERSION : 0.1
   VAR_TEMP   // added for the SCL form of the ladder/FBD networks
      _w1 : Bool;
   END_VAR
BEGIN

REGION Network 2: =================Блокування пристрою ручного керування========================
END_REGION

REGION Network 3: Механізм пересування крана. Дозвіл роботи (РП роз'єднан з приводом). 4SQ41
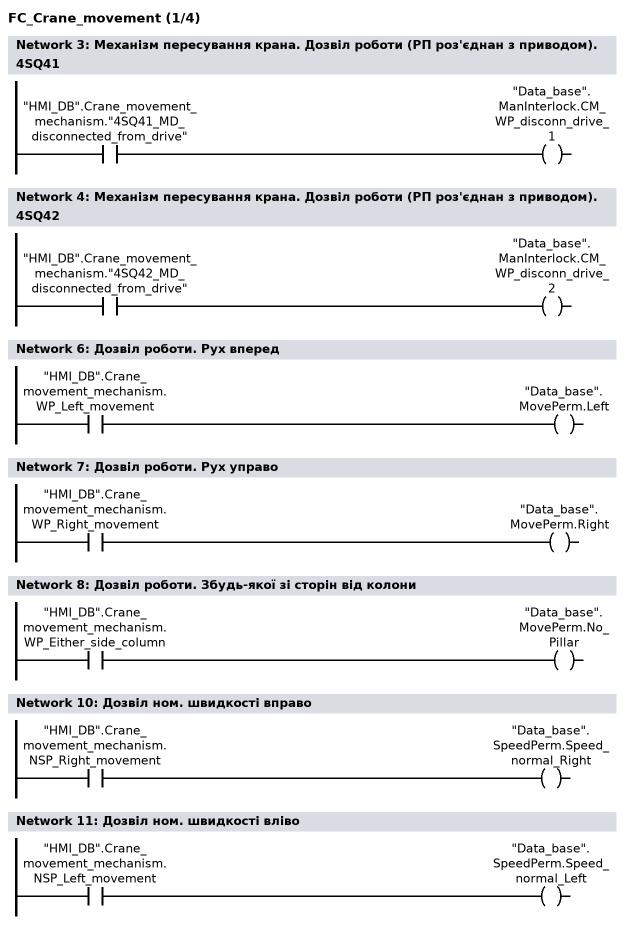
   RUNG wire#powerrail
      Contact( "HMI_DB".Crane_movement_mechanism."4SQ41_MD_disconnected_from_drive" )
      Coil( "Data_base".ManInterlock.CM_WP_disconn_drive_1 )
   END_RUNG
   // the same network as SCL:
   "Data_base".ManInterlock.CM_WP_disconn_drive_1 := "HMI_DB".Crane_movement_mechanism."4SQ41_MD_disconnected_from_drive";
END_REGION

REGION Network 4: Механізм пересування крана. Дозвіл роботи (РП роз'єднан з приводом). 4SQ42
   RUNG wire#powerrail
      Contact( "HMI_DB".Crane_movement_mechanism."4SQ42_MD_disconnected_from_drive" )
      Coil( "Data_base".ManInterlock.CM_WP_disconn_drive_2 )
   END_RUNG
   // the same network as SCL:
   "Data_base".ManInterlock.CM_WP_disconn_drive_2 := "HMI_DB".Crane_movement_mechanism."4SQ42_MD_disconnected_from_drive";
END_REGION

REGION Network 5: ================Дозвіл роботи====================
END_REGION

REGION Network 6: Дозвіл роботи. Рух вперед
   RUNG wire#powerrail
      Contact( "HMI_DB".Crane_movement_mechanism.WP_Left_movement )
      Coil( "Data_base".MovePerm.Left )
   END_RUNG
   // the same network as SCL:
   "Data_base".MovePerm.Left := "HMI_DB".Crane_movement_mechanism.WP_Left_movement;
END_REGION

REGION Network 7: Дозвіл роботи. Рух управо
   RUNG wire#powerrail
      Contact( "HMI_DB".Crane_movement_mechanism.WP_Right_movement )
      Coil( "Data_base".MovePerm.Right )
   END_RUNG
   // the same network as SCL:
   "Data_base".MovePerm.Right := "HMI_DB".Crane_movement_mechanism.WP_Right_movement;
END_REGION

REGION Network 8: Дозвіл роботи. Збудь-якої зі сторін від колони
   RUNG wire#powerrail
      Contact( "HMI_DB".Crane_movement_mechanism.WP_Either_side_column )
      Coil( "Data_base".MovePerm.No_Pillar )
   END_RUNG
   // the same network as SCL:
   "Data_base".MovePerm.No_Pillar := "HMI_DB".Crane_movement_mechanism.WP_Either_side_column;
END_REGION

REGION Network 9: ================Дозвіл нормальної швидкості =================
END_REGION

REGION Network 10: Дозвіл ном. швидкості вправо
   RUNG wire#powerrail
      Contact( "HMI_DB".Crane_movement_mechanism.NSP_Right_movement )
      Coil( "Data_base".SpeedPerm.Speed_normal_Right )
   END_RUNG
   // the same network as SCL:
   "Data_base".SpeedPerm.Speed_normal_Right := "HMI_DB".Crane_movement_mechanism.NSP_Right_movement;
END_REGION

REGION Network 11: Дозвіл ном. швидкості вліво
   RUNG wire#powerrail
      Contact( "HMI_DB".Crane_movement_mechanism.NSP_Left_movement )
      Coil( "Data_base".SpeedPerm.Speed_normal_Left )
   END_RUNG
   // the same network as SCL:
   "Data_base".SpeedPerm.Speed_normal_Left := "HMI_DB".Crane_movement_mechanism.NSP_Left_movement;
END_REGION

REGION Network 12: ===============Керування механізмом крана================ / ===============Керування механізмом підйому================
END_REGION

